KUKA KRL program: MyProgram_314().src

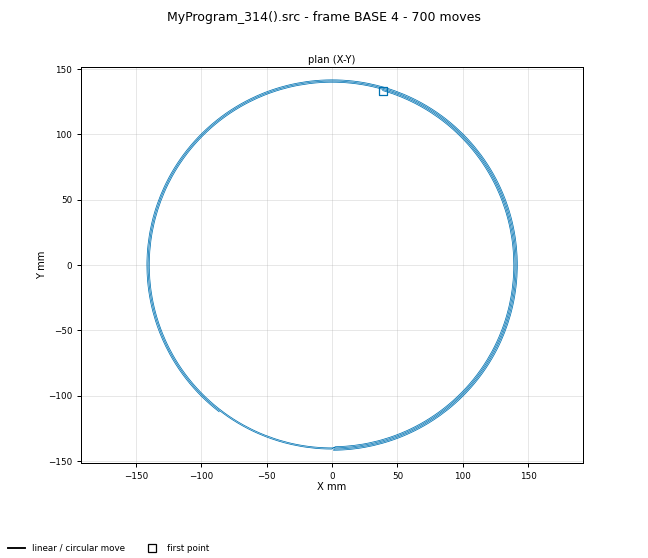
[picture p0: tool path of MyProgram_314().src in frame BASE 4, 700 of 700 moves have a stored position in this frame; points joined in program order, loops and branches not executed]
&ACCESS RVP
&REL 1
&PARAM TEMPLATE = C:\KRC\Roboter\Template\vorgabe
&PARAM EDITMASK = *
DEF MyProgram_314()
; ---- Setting reference (Base) ----
$BASE = BASE_DATA[4]

; --------------------------
; ---- Setting tool (TCP) ----
$TOOL = TOOL_DATA[3]
; --------------------------

$VEL.CP = VEL_APROX_PRINT
Startdeposition()
$VEL.CP = VEL_PRINT
LIN {X 38.6901,Y 133.5484,Z 183,A 74.6079,B 4.1647,C 0.0823,E1 4.2136,E2 378.5903} C_DIS
LIN {X 41.5849,Y 132.6771,Z 183,A 73.3895,B 4.1647,C 0.0831,E1 4.2168,E2 379.8051} C_DIS
LIN {X 46.4124,Y 131.0665,Z 183,A 71.2167,B 4.1647,C 0.0859,E1 4.2226,E2 381.9869} C_DIS
LIN {X 50.1301,Y 129.6879,Z 183,A 69.6295,B 4.1646,C 0.0872,E1 4.2267,E2 383.568} C_DIS
LIN {X 53.3488,Y 128.3973,Z 183,A 68.1306,B 4.1646,C 0.0895,E1 4.2306,E2 385.0754} C_DIS
LIN {X 57.8954,Y 126.4131,Z 183,A 65.4479,B 4.1643,C 0.0987,E1 4.2376,E2 387.8363} C_DIS
LIN {X 63.5941,Y 123.6447,Z 183,A 63.5677,B 4.1644,C 0.0945,E1 4.2421,E2 389.6266} C_DIS
LIN {X 67.8619,Y 121.3561,Z 183,A 61.634,B 4.1644,C 0.0967,E1 4.2468,E2 391.5526} C_DIS
LIN {X 71.8304,Y 119.0499,Z 183,A 59.745,B 4.1644,C 0.0995,E1 4.2513,E2 393.4412} C_DIS
LIN {X 75.3981,Y 116.8235,Z 183,A 58.2199,B 4.1644,C 0.1,E1 4.2549,E2 394.9405} C_DIS
LIN {X 81.6488,Y 112.543,Z 183,A 55.058,B 4.1642,C 0.1056,E1 4.2622,E2 398.1075} C_DIS
LIN {X 85.258,Y 109.8341,Z 183,A 53.2155,B 4.1641,C 0.1087,E1 4.2662,E2 399.948} C_DIS
LIN {X 88.7432,Y 107.0378,Z 183,A 51.4298,B 4.1641,C 0.1114,E1 4.2701,E2 401.727} C_DIS
LIN {X 92.1738,Y 104.0983,Z 183,A 49.6505,B 4.1639,C 0.114,E1 4.2738,E2 403.4963} C_DIS
LIN {X 95.5936,Y 100.9672,Z 183,A 47.5183,B 4.1638,C 0.1203,E1 4.2782,E2 405.6563} C_DIS
LIN {X 98.0318,Y 98.6013,Z 183,A 46.3699,B 4.1638,C 0.1203,E1 4.2805,E2 406.7736} C_DIS
LIN {X 101.2747,Y 95.2677,Z 183,A 44.4916,B 4.1637,C 0.1238,E1 4.2841,E2 408.6476} C_DIS
LIN {X 104.2938,Y 91.9527,Z 183,A 42.7466,B 4.1636,C 0.1266,E1 4.2873,E2 410.3801} C_DIS
LIN {X 107.0493,Y 88.7294,Z 183,A 41.1805,B 4.1636,C 0.1283,E1 4.2901,E2 411.9238} C_DIS
LIN {X 109.6954,Y 85.4369,Z 183,A 39.261,B 4.1633,C 0.1343,E1 4.2935,E2 413.8663} C_DIS
LIN {X 112.5064,Y 81.6994,Z 183,A 37.4355,B 4.1633,C 0.1375,E1 4.2965,E2 415.6797} C_DIS
LIN {X 115.0062,Y 78.1414,Z 183,A 35.6994,B 4.1631,C 0.1411,E1 4.2992,E2 417.4092} C_DIS
LIN {X 117.403,Y 74.4922,Z 183,A 33.895,B 4.163,C 0.1454,E1 4.302,E2 419.2149} C_DIS
LIN {X 119.858,Y 70.4735,Z 183,A 32.0698,B 4.1628,C 0.1488,E1 4.3046,E2 421.0263} C_DIS
LIN {X 121.9501,Y 66.7885,Z 183,A 30.3317,B 4.1627,C 0.153,E1 4.3069,E2 422.7641} C_DIS
LIN {X 123.8361,Y 63.2182,Z 183,A 28.7952,B 4.1626,C 0.1557,E1 4.3089,E2 424.285} C_DIS
LIN {X 125.6527,Y 59.5273,Z 183,A 27.0862,B 4.1624,C 0.1602,E1 4.311,E2 425.9966} C_DIS
LIN {X 127.4768,Y 55.5132,Z 183,A 25.4211,B 4.1624,C 0.1631,E1 4.3128,E2 427.6432} C_DIS
LIN {X 128.8068,Y 52.3534,Z 183,A 24.0226,B 4.1622,C 0.1666,E1 4.3143,E2 429.0406} C_DIS
LIN {X 130.1139,Y 49.0137,Z 183,A 22.5912,B 4.162,C 0.17,E1 4.3158,E2 430.4669} C_DIS
LIN {X 131.3645,Y 45.5554,Z 183,A 21.1712,B 4.162,C 0.1728,E1 4.3171,E2 431.8754} C_DIS
LIN {X 132.3962,Y 42.4643,Z 183,A 19.8538,B 4.1618,C 0.1762,E1 4.3182,E2 433.1903} C_DIS
LIN {X 133.3699,Y 39.2998,Z 183,A 18.6395,B 4.1618,C 0.178,E1 4.3192,E2 434.3862} C_DIS
LIN {X 134.5526,Y 35.0458,Z 183,A 16.6466,B 4.1614,C 0.1851,E1 4.3207,E2 436.4024} C_DIS
LIN {X 135.5223,Y 31.0755,Z 183,A 15.1454,B 4.1613,C 0.1875,E1 4.3216,E2 437.8811} C_DIS
LIN {X 136.2197,Y 27.8599,Z 183,A 13.8266,B 4.1611,C 0.1908,E1 4.3224,E2 439.1959} C_DIS
LIN {X 137.5207,Y 20.5096,Z 183,A 10.874,B 4.1608,C 0.1979,E1 4.3238,E2 442.1347} C_DIS
LIN {X 137.9086,Y 17.7021,Z 183,A 9.3425,B 4.1604,C 0.2057,E1 4.3243,E2 443.7134} C_DIS
LIN {X 138.3551,Y 13.7893,Z 183,A 8.0826,B 4.1604,C 0.2057,E1 4.3247,E2 444.9281} C_DIS
LIN {X 138.6565,Y 10.3177,Z 183,A 6.7452,B 4.1603,C 0.2086,E1 4.325,E2 446.2537} C_DIS
LIN {X 138.8833,Y 6.6033,Z 183,A 5.211,B 4.1601,C 0.2129,E1 4.3252,E2 447.7891} C_DIS
LIN {X 139.0156,Y 2.6101,Z 183,A 3.8011,B 4.16,C 0.2146,E1 4.3252,E2 449.1697} C_DIS
LIN {X 139.0434,Y -0.021,Z 183,A 2.504,B 4.1597,C 0.2204,E1 4.3253,E2 450.495} C_DIS
LIN {X 138.9836,Y -3.952,Z 183,A 1.081,B 4.1596,C 0.2225,E1 4.3253,E2 451.8937} C_DIS
LIN {X 138.8076,Y -8.0465,Z 183,A -0.5936,B 4.1593,C 0.2271,E1 4.325,E2 453.5677} C_DIS
LIN {X 138.5359,Y -11.8261,Z 183,A -2.0469,B 4.1591,C 0.2301,E1 4.3247,E2 455.0081} C_DIS
LIN {X 138.1515,Y -15.7085,Z 183,A -3.7013,B 4.1589,C 0.2353,E1 4.3242,E2 456.6699} C_DIS
LIN {X 137.76,Y -18.8356,Z 183,A -5.4114,B 4.1584,C 0.2441,E1 4.3235,E2 458.434} C_DIS
LIN {X 137.0345,Y -23.5365,Z 183,A -6.7142,B 4.1585,C 0.2414,E1 4.323,E2 459.6534} C_DIS
LIN {X 135.6633,Y -30.4582,Z 183,A -9.607,B 4.158,C 0.2493,E1 4.3214,E2 462.5467} C_DIS
LIN {X 134.9201,Y -33.5994,Z 183,A -11.0898,B 4.1577,C 0.2549,E1 4.3203,E2 464.0503} C_DIS
LIN {X 133.5628,Y -38.6411,Z 183,A -12.8026,B 4.1577,C 0.2553,E1 4.3191,E2 465.7078} C_DIS
LIN {X 132.6254,Y -41.7467,Z 183,A -14.2307,B 4.1574,C 0.2601,E1 4.3179,E2 467.1489} C_DIS
LIN {X 131.4955,Y -45.1776,Z 183,A -16.076,B 4.1569,C 0.2685,E1 4.3162,E2 469.0418} C_DIS
LIN {X 130.171,Y -48.8614,Z 183,A -17.2495,B 4.1569,C 0.2674,E1 4.3152,E2 470.1594} C_DIS
LIN {X 128.9622,Y -51.9679,Z 183,A -18.5228,B 4.1568,C 0.2698,E1 4.3139,E2 471.4208} C_DIS
LIN {X 127.7218,Y -54.9464,Z 183,A -19.807,B 4.1566,C 0.2728,E1 4.3125,E2 472.7002} C_DIS
LIN {X 125.9756,Y -58.8415,Z 183,A -21.66,B 4.1562,C 0.2785,E1 4.3103,E2 474.5669} C_DIS
LIN {X 124.2812,Y -62.3432,Z 183,A -23.2186,B 4.156,C 0.2821,E1 4.3084,E2 476.1211} C_DIS
LIN {X 122.3977,Y -65.9643,Z 183,A -24.8332,B 4.1557,C 0.2855,E1 4.3063,E2 477.7283} C_DIS
LIN {X 118.702,Y -72.4046,Z 183,A -27.8541,B 4.1552,C 0.2927,E1 4.302,E2 480.7467} C_DIS
LIN {X 116.1898,Y -76.3701,Z 183,A -29.6676,B 4.155,C 0.2959,E1 4.2993,E2 482.546} C_DIS
LIN {X 113.7481,Y -79.9617,Z 183,A -31.4516,B 4.1547,C 0.3001,E1 4.2965,E2 484.3308} C_DIS
LIN {X 111.0357,Y -83.6871,Z 183,A -33.2889,B 4.1544,C 0.3038,E1 4.2934,E2 486.1616} C_DIS
LIN {X 108.1883,Y -87.337,Z 183,A -35.1586,B 4.1541,C 0.3077,E1 4.2902,E2 488.0279} C_DIS
LIN {X 105.1296,Y -90.9963,Z 183,A -37.0564,B 4.1539,C 0.3112,E1 4.2868,E2 489.9184} C_DIS
LIN {X 102.0998,Y -94.3835,Z 183,A -38.8813,B 4.1536,C 0.3147,E1 4.2833,E2 491.7386} C_DIS
LIN {X 99.1255,Y -97.5019,Z 183,A -40.6699,B 4.1533,C 0.3186,E1 4.2799,E2 493.5304} C_DIS
LIN {X 95.672,Y -100.8932,Z 183,A -42.5669,B 4.1531,C 0.3215,E1 4.2761,E2 495.4161} C_DIS
LIN {X 92.5142,Y -103.7964,Z 183,A -44.2085,B 4.1529,C 0.3236,E1 4.2727,E2 497.0426} C_DIS
LIN {X 89.4317,Y -106.4633,Z 183,A -45.9892,B 4.1526,C 0.328,E1 4.2689,E2 498.838} C_DIS
LIN {X 85.6496,Y -109.5294,Z 183,A -47.8402,B 4.1524,C 0.3299,E1 4.2649,E2 500.6701} C_DIS
LIN {X 82.2654,Y -112.0931,Z 183,A -49.5595,B 4.1522,C 0.3327,E1 4.261,E2 502.3869} C_DIS
LIN {X 78.6574,Y -114.6537,Z 183,A -51.3807,B 4.152,C 0.3358,E1 4.2569,E2 504.2092} C_DIS
LIN {X 74.8249,Y -117.191,Z 183,A -53.2055,B 4.1518,C 0.3381,E1 4.2526,E2 506.0263} C_DIS
LIN {X 71.0409,Y -119.5227,Z 183,A -54.9847,B 4.1516,C 0.3404,E1 4.2484,E2 507.7999} C_DIS
LIN {X 67.9317,Y -121.3169,Z 183,A -56.5366,B 4.1513,C 0.3434,E1 4.2446,E2 509.3626} C_DIS
LIN {X 63.7821,Y -123.549,Z 183,A -58.4038,B 4.1512,C 0.3454,E1 4.24,E2 511.2214} C_DIS
LIN {X 60.2118,Y -125.3257,Z 183,A -59.9855,B 4.1511,C 0.3469,E1 4.236,E2 512.7961} C_DIS
LIN {X 57.1271,Y -126.7618,Z 183,A -61.3521,B 4.1509,C 0.3484,E1 4.2326,E2 514.159} C_DIS
LIN {X 52.8925,Y -128.5879,Z 183,A -63.2697,B 4.1507,C 0.3509,E1 4.2276,E2 516.0803} C_DIS
LIN {X 48.2273,Y -130.4085,Z 183,A -65.6657,B 4.1502,C 0.3568,E1 4.2212,E2 518.5216} C_DIS
LIN {X 44.2524,Y -131.8096,Z 183,A -66.9438,B 4.1505,C 0.3537,E1 4.218,E2 519.7401} C_DIS
LIN {X 41.1074,Y -132.8244,Z 183,A -68.3125,B 4.1504,C 0.3551,E1 4.2144,E2 521.1107} C_DIS
LIN {X 38.0143,Y -133.7431,Z 183,A -69.6747,B 4.1502,C 0.3566,E1 4.2107,E2 522.4781} C_DIS
LIN {X 34.8764,Y -134.596,Z 183,A -71.3347,B 4.1498,C 0.3611,E1 4.2061,E2 524.1815} C_DIS
LIN {X 31.0318,Y -135.5323,Z 183,A -72.5205,B 4.1501,C 0.3578,E1 4.203,E2 525.3093} C_DIS
LIN {X 27.8154,Y -136.2288,Z 183,A -73.7669,B 4.1501,C 0.3576,E1 4.1997,E2 526.5418} C_DIS
LIN {X 23.5961,Y -137.0246,Z 183,A -75.5986,B 4.15,C 0.3594,E1 4.1946,E2 528.383} C_DIS
LIN {X 16.847,Y -138.0157,Z 183,A -78.445,B 4.1498,C 0.3612,E1 4.1867,E2 531.2357} C_DIS
LIN {X 13.4116,Y -138.3913,Z 183,A -79.7844,B 4.1498,C 0.361,E1 4.183,E2 532.5645} C_DIS
LIN {X 10.2776,Y -138.6594,Z 183,A -81.1632,B 4.1498,C 0.3623,E1 4.1791,E2 533.9551} C_DIS
LIN {X 6.3212,Y -138.8975,Z 183,A -82.7609,B 4.1498,C 0.3624,E1 4.1747,E2 535.5489} C_DIS
LIN {X 2.5424,Y -139.0167,Z 183,A -84.3219,B 4.1498,C 0.3628,E1 4.1703,E2 537.111} C_DIS
LIN {X 2.5424,Y -139.0167,Z 183,A -84.3219,B 4.1498,C 0.3628,E1 4.1703,E2 537.111} C_DIS
Enddeposition()
LIN {X 0.9796,Y -139.9354,Z 183,A -84.7324,B 4.1032,C 0.3616,E1 4.1227,E2 537.5356} C_DIS
Startdeposition()
$VEL.CP = VEL_PRINT
LIN {X 3.736,Y -139.891,Z 183,A -83.0903,B 4.1037,C 0.3563,E1 4.1275,E2 535.8237} C_DIS
LIN {X 7.4249,Y -139.7442,Z 183,A -81.5162,B 4.1037,C 0.3553,E1 4.1319,E2 534.2403} C_DIS
LIN {X 11.7645,Y -139.4453,Z 183,A -79.8462,B 4.1037,C 0.3557,E1 4.1365,E2 532.5844} C_DIS
LIN {X 15.3477,Y -139.097,Z 183,A -78.4152,B 4.1037,C 0.3555,E1 4.1405,E2 531.1584} C_DIS
LIN {X 18.9985,Y -138.6472,Z 183,A -76.606,B 4.1041,C 0.3517,E1 4.1456,E2 529.3073} C_DIS
LIN {X 22.2848,Y -138.1565,Z 183,A -75.599,B 4.1038,C 0.3545,E1 4.1482,E2 528.3475} C_DIS
LIN {X 28.614,Y -136.9858,Z 183,A -72.9607,B 4.104,C 0.3528,E1 4.1555,E2 525.7073} C_DIS
LIN {X 31.4563,Y -136.3595,Z 183,A -71.592,B 4.1042,C 0.35,E1 4.1593,E2 524.3138} C_DIS
LIN {X 36.5456,Y -135.0851,Z 183,A -69.6426,B 4.1042,C 0.3503,E1 4.1645,E2 522.3901} C_DIS
LIN {X 39.5732,Y -134.2287,Z 183,A -68.346,B 4.1043,C 0.349,E1 4.168,E2 521.0915} C_DIS
LIN {X 43.4113,Y -133.0393,Z 183,A -66.4686,B 4.1047,C 0.3449,E1 4.1731,E2 519.1815} C_DIS
LIN {X 49.2904,Y -130.9725,Z 183,A -64.2268,B 4.1046,C 0.3455,E1 4.1788,E2 516.9799} C_DIS
LIN {X 52.381,Y -129.7671,Z 183,A -62.8427,B 4.1048,C 0.3436,E1 4.1824,E2 515.5914} C_DIS
LIN {X 55.7191,Y -128.3694,Z 183,A -61.4245,B 4.1048,C 0.3425,E1 4.1861,E2 514.1807} C_DIS
LIN {X 59.1512,Y -126.8251,Z 183,A -59.8958,B 4.105,C 0.3406,E1 4.19,E2 512.6526} C_DIS
LIN {X 62.3488,Y -125.2842,Z 183,A -58.4371,B 4.1052,C 0.3386,E1 4.1936,E2 511.192} C_DIS
LIN {X 66.3568,Y -123.2097,Z 183,A -56.3022,B 4.1057,C 0.3327,E1 4.199,E2 509.0168} C_DIS
LIN {X 69.5862,Y -121.4151,Z 183,A -55.0814,B 4.1056,C 0.3337,E1 4.2019,E2 507.8345} C_DIS
LIN {X 73.4646,Y -119.1087,Z 183,A -53.2489,B 4.1058,C 0.331,E1 4.2062,E2 506.0026} C_DIS
LIN {X 77.1485,Y -116.7561,Z 183,A -51.2986,B 4.1062,C 0.3262,E1 4.2109,E2 504.0291} C_DIS
LIN {X 79.9664,Y -114.8443,Z 183,A -49.7608,B 4.1065,C 0.3221,E1 4.2144,E2 502.4707} C_DIS
LIN {X 83.5364,Y -112.2742,Z 183,A -48.745,B 4.106,C 0.3281,E1 4.2165,E2 501.5598} C_DIS
LIN {X 87.4834,Y -109.2276,Z 183,A -46.0047,B 4.107,C 0.3161,E1 4.2227,E2 498.7234} C_DIS
LIN {X 90.836,Y -106.4551,Z 183,A -44.2671,B 4.1072,C 0.3132,E1 4.2264,E2 496.9903} C_DIS
LIN {X 94.111,Y -103.571,Z 183,A -42.8999,B 4.1071,C 0.3147,E1 4.2291,E2 495.6784} C_DIS
LIN {X 97.4757,Y -100.4109,Z 183,A -40.7399,B 4.1076,C 0.3076,E1 4.2335,E2 493.4803} C_DIS
LIN {X 100.3317,Y -97.5575,Z 183,A -39.3383,B 4.1076,C 0.3071,E1 4.2362,E2 492.1114} C_DIS
LIN {X 103.6153,Y -94.0622,Z 183,A -37.5343,B 4.1078,C 0.3048,E1 4.2396,E2 490.3272} C_DIS
LIN {X 106.5619,Y -90.7105,Z 183,A -35.7303,B 4.1081,C 0.3011,E1 4.2429,E2 488.5248} C_DIS
LIN {X 108.8719,Y -87.9247,Z 183,A -34.301,B 4.1083,C 0.2984,E1 4.2454,E2 487.1013} C_DIS
LIN {X 111.7372,Y -84.2533,Z 183,A -32.4639,B 4.1085,C 0.2948,E1 4.2485,E2 485.272} C_DIS
LIN {X 114.4356,Y -80.5502,Z 183,A -30.6302,B 4.1088,C 0.2909,E1 4.2515,E2 483.4424} C_DIS
LIN {X 117.0012,Y -76.7762,Z 183,A -28.8143,B 4.1091,C 0.2871,E1 4.2543,E2 481.632} C_DIS
LIN {X 119.43,Y -72.941,Z 183,A -26.8652,B 4.1095,C 0.2814,E1 4.2572,E2 479.6691} C_DIS
LIN {X 122.7694,Y -67.168,Z 183,A -24.2566,B 4.1098,C 0.2761,E1 4.2607,E2 477.0746} C_DIS
LIN {X 124.8058,Y -63.2994,Z 183,A -22.7216,B 4.1099,C 0.2746,E1 4.2627,E2 475.5722} C_DIS
LIN {X 126.202,Y -60.4677,Z 183,A -21.0647,B 4.1105,C 0.2668,E1 4.2647,E2 473.8654} C_DIS
LIN {X 127.8914,Y -56.8084,Z 183,A -19.8668,B 4.1104,C 0.2681,E1 4.266,E2 472.7267} C_DIS
LIN {X 129.2282,Y -53.6973,Z 183,A -18.5019,B 4.1106,C 0.2647,E1 4.2675,E2 471.3635} C_DIS
LIN {X 130.534,Y -50.4403,Z 183,A -17.1692,B 4.1107,C 0.2622,E1 4.2688,E2 470.0435} C_DIS
LIN {X 132.5502,Y -44.8802,Z 183,A -14.7377,B 4.1112,C 0.2556,E1 4.2711,E2 467.6087} C_DIS
LIN {X 133.7534,Y -41.1506,Z 183,A -13.1595,B 4.1114,C 0.2515,E1 4.2724,E2 466.0326} C_DIS
LIN {X 134.9002,Y -37.222,Z 183,A -10.8806,B 4.1121,C 0.2393,E1 4.2742,E2 463.6718} C_DIS
LIN {X 136.3491,Y -31.5022,Z 183,A -9.3294,B 4.1119,C 0.2435,E1 4.2751,E2 462.2341} C_DIS
LIN {X 137.6457,Y -25.2466,Z 183,A -6.8343,B 4.1122,C 0.2378,E1 4.2765,E2 459.7531} C_DIS
LIN {X 138.1132,Y -22.5464,Z 183,A -5.5729,B 4.1125,C 0.2329,E1 4.2771,E2 458.4724} C_DIS
LIN {X 138.6569,Y -18.9261,Z 183,A -4.2506,B 4.1126,C 0.2309,E1 4.2776,E2 457.1723} C_DIS
LIN {X 139.1517,Y -14.8395,Z 183,A -2.5527,B 4.1129,C 0.226,E1 4.2781,E2 455.4715} C_DIS
LIN {X 139.5467,Y -10.4986,Z 183,A -0.8139,B 4.1131,C 0.2215,E1 4.2785,E2 453.7373} C_DIS
LIN {X 139.7795,Y -6.7232,Z 183,A 0.6384,B 4.1133,C 0.2183,E1 4.2788,E2 452.2967} C_DIS
LIN {X 139.8999,Y -3.4143,Z 183,A 2.0229,B 4.1135,C 0.2141,E1 4.2788,E2 450.9073} C_DIS
LIN {X 139.9405,Y 0.6341,Z 183,A 3.6219,B 4.1137,C 0.2102,E1 4.2788,E2 449.315} C_DIS
LIN {X 139.8518,Y 5.0079,Z 183,A 5.3432,B 4.1139,C 0.206,E1 4.2788,E2 447.6016} C_DIS
LIN {X 139.658,Y 8.895,Z 183,A 6.8354,B 4.1141,C 0.2027,E1 4.2785,E2 446.1216} C_DIS
LIN {X 139.3232,Y 13.1336,Z 183,A 8.5685,B 4.1143,C 0.1979,E1 4.2781,E2 444.3883} C_DIS
LIN {X 138.769,Y 18.0706,Z 183,A 10.4614,B 4.1145,C 0.194,E1 4.2775,E2 442.5126} C_DIS
LIN {X 138.2844,Y 21.4663,Z 183,A 12.454,B 4.115,C 0.1827,E1 4.2766,E2 440.4419} C_DIS
LIN {X 137.365,Y 26.7287,Z 183,A 14.253,B 4.115,C 0.1815,E1 4.2757,E2 438.6927} C_DIS
LIN {X 136.6393,Y 30.2249,Z 183,A 15.3384,B 4.115,C 0.1821,E1 4.2751,E2 437.6557} C_DIS
LIN {X 135.9274,Y 33.2762,Z 183,A 16.5818,B 4.1152,C 0.1791,E1 4.2742,E2 436.4166} C_DIS
LIN {X 134.5668,Y 38.4144,Z 183,A 18.6873,B 4.1154,C 0.174,E1 4.2727,E2 434.3192} C_DIS
LIN {X 133.7792,Y 41.0662,Z 183,A 19.8093,B 4.1155,C 0.171,E1 4.2718,E2 433.198} C_DIS
LIN {X 132.7549,Y 44.2656,Z 183,A 21.1119,B 4.1157,C 0.1682,E1 4.2707,E2 431.9041} C_DIS
LIN {X 131.6037,Y 47.579,Z 183,A 22.5424,B 4.1158,C 0.1645,E1 4.2693,E2 430.4736} C_DIS
LIN {X 130.3743,Y 50.8513,Z 183,A 23.9233,B 4.1159,C 0.1613,E1 4.268,E2 429.0985} C_DIS
LIN {X 129.0654,Y 54.0872,Z 183,A 25.3216,B 4.1161,C 0.1579,E1 4.2665,E2 427.7035} C_DIS
LIN {X 127.6068,Y 57.4446,Z 183,A 26.7566,B 4.1161,C 0.1548,E1 4.2649,E2 426.2761} C_DIS
LIN {X 126.1331,Y 60.6118,Z 183,A 28.142,B 4.1163,C 0.1517,E1 4.2632,E2 424.8959} C_DIS
LIN {X 124.5227,Y 63.8554,Z 183,A 29.5799,B 4.1164,C 0.1485,E1 4.2614,E2 423.4631} C_DIS
LIN {X 122.717,Y 67.2641,Z 183,A 31.2028,B 4.1166,C 0.144,E1 4.2593,E2 421.834} C_DIS
LIN {X 120.4869,Y 71.1818,Z 183,A 32.974,B 4.1167,C 0.1403,E1 4.2568,E2 420.0718} C_DIS
LIN {X 118.1588,Y 74.983,Z 183,A 34.7723,B 4.1168,C 0.1363,E1 4.2541,E2 418.2762} C_DIS
LIN {X 115.6435,Y 78.8073,Z 183,A 36.5684,B 4.117,C 0.1327,E1 4.2514,E2 416.4896} C_DIS
LIN {X 113.0942,Y 82.4236,Z 183,A 38.3345,B 4.117,C 0.1291,E1 4.2485,E2 414.7287} C_DIS
LIN {X 110.4665,Y 85.9129,Z 183,A 40.5753,B 4.1174,C 0.1197,E1 4.2446,E2 412.4291} C_DIS
LIN {X 107.2942,Y 89.8431,Z 183,A 42.0484,B 4.1173,C 0.1221,E1 4.2421,E2 411.0322} C_DIS
LIN {X 104.498,Y 93.0813,Z 183,A 43.8953,B 4.1174,C 0.1172,E1 4.2386,E2 409.1727} C_DIS
LIN {X 101.654,Y 96.1786,Z 183,A 45.463,B 4.1174,C 0.1154,E1 4.2357,E2 407.6243} C_DIS
LIN {X 98.5993,Y 99.3076,Z 183,A 47.8184,B 4.1177,C 0.1053,E1 4.2309,E2 405.196} C_DIS
LIN {X 94.5364,Y 103.1831,Z 183,A 49.3534,B 4.1177,C 0.1095,E1 4.2279,E2 403.7587} C_DIS
LIN {X 92.1545,Y 105.3158,Z 183,A 50.7655,B 4.1177,C 0.1058,E1 4.2249,E2 402.3333} C_DIS
LIN {X 88.3263,Y 108.5466,Z 183,A 52.7567,B 4.1178,C 0.1027,E1 4.2207,E2 400.3495} C_DIS
LIN {X 84.6897,Y 111.4076,Z 183,A 54.6308,B 4.1178,C 0.0996,E1 4.2165,E2 398.4779} C_DIS
LIN {X 80.7626,Y 114.2855,Z 183,A 56.794,B 4.118,C 0.0943,E1 4.2116,E2 396.2929} C_DIS
LIN {X 77.8149,Y 116.3129,Z 183,A 57.9478,B 4.118,C 0.0953,E1 4.209,E2 395.1787} C_DIS
LIN {X 74.2993,Y 118.5902,Z 183,A 59.7134,B 4.118,C 0.0921,E1 4.2048,E2 393.4066} C_DIS
LIN {X 70.6261,Y 120.8133,Z 183,A 61.3857,B 4.118,C 0.0904,E1 4.2008,E2 391.7453} C_DIS
LIN {X 66.6812,Y 123.0349,Z 183,A 63.2276,B 4.1182,C 0.0879,E1 4.1963,E2 389.9049} C_DIS
LIN {X 62.8771,Y 125.0208,Z 183,A 65.1802,B 4.1182,C 0.0834,E1 4.1914,E2 387.9276} C_DIS
LIN {X 59.7314,Y 126.5537,Z 183,A 66.2498,B 4.1182,C 0.0854,E1 4.1888,E2 386.9042} C_DIS
LIN {X 57.0233,Y 127.7953,Z 183,A 67.4511,B 4.1182,C 0.0841,E1 4.1858,E2 385.7053} C_DIS
LIN {X 53.6698,Y 129.2397,Z 183,A 68.9309,B 4.1182,C 0.0825,E1 4.182,E2 384.2277} C_DIS
LIN {X 50.4125,Y 130.5449,Z 183,A 70.3823,B 4.1182,C 0.0808,E1 4.1782,E2 382.7746} C_DIS
LIN {X 46.7659,Y 131.8969,Z 183,A 72.6408,B 4.1185,C 0.0724,E1 4.172,E2 380.4319} C_DIS
LIN {X 41.4513,Y 133.6614,Z 183,A 74.0818,B 4.1183,C 0.0789,E1 4.1685,E2 379.0994} C_DIS
LIN {X 38.9881,Y 134.4,Z 183,A 75.2244,B 4.1183,C 0.0771,E1 4.1654,E2 377.9458} C_DIS
LIN {X 35.4655,Y 135.3732,Z 183,A 76.9224,B 4.1184,C 0.0739,E1 4.1607,E2 376.2226} C_DIS
LIN {X 31.1573,Y 136.4278,Z 183,A 78.8391,B 4.1184,C 0.0716,E1 4.1555,E2 374.2936} C_DIS
LIN {X 27.7717,Y 137.1572,Z 183,A 79.9625,B 4.1184,C 0.0735,E1 4.1525,E2 373.2078} C_DIS
LIN {X 23.9362,Y 137.8802,Z 183,A 81.8001,B 4.1184,C 0.0703,E1 4.1474,E2 371.3406} C_DIS
LIN {X 18.614,Y 138.6978,Z 183,A 83.5571,B 4.1184,C 0.0735,E1 4.1427,E2 369.6406} C_DIS
LIN {X 14.7295,Y 139.1635,Z 183,A 85.3706,B 4.1184,C 0.0709,E1 4.1376,E2 367.8011} C_DIS
LIN {X 10.3429,Y 139.558,Z 183,A 87.1238,B 4.1184,C 0.0709,E1 4.1327,E2 366.0549} C_DIS
LIN {X 6.8393,Y 139.7736,Z 183,A 88.5411,B 4.1184,C 0.0707,E1 4.1288,E2 364.6407} C_DIS
LIN {X 2.8571,Y 139.9126,Z 183,A 90.2468,B 4.1184,C 0.0697,E1 4.124,E2 362.9263} C_DIS
LIN {X -1.1552,Y 139.9366,Z 183,A 91.7864,B 4.1184,C 0.0705,E1 4.1197,E2 361.4004} C_DIS
LIN {X -4.9256,Y 139.855,Z 183,A 93.4859,B 4.1185,C 0.0691,E1 4.1149,E2 359.6821} C_DIS
LIN {X -8.937,Y 139.6555,Z 183,A 95.167,B 4.1185,C 0.069,E1 4.1102,E2 357.9971} C_DIS
LIN {X -12.5685,Y 139.3774,Z 183,A 96.6629,B 4.1185,C 0.0692,E1 4.106,E2 356.5014} C_DIS
LIN {X -16.9807,Y 138.9072,Z 183,A 98.3677,B 4.1185,C 0.0706,E1 4.1013,E2 354.8115} C_DIS
LIN {X -25.8176,Y 137.5391,Z 183,A 102.1653,B 4.1185,C 0.0709,E1 4.0908,E2 350.9989} C_DIS
LIN {X -30.0571,Y 136.6755,Z 183,A 103.765,B 4.1185,C 0.0732,E1 4.0865,E2 349.4219} C_DIS
LIN {X -33.2613,Y 135.931,Z 183,A 105.2627,B 4.1185,C 0.0727,E1 4.0824,E2 347.906} C_DIS
LIN {X -39.3908,Y 134.2821,Z 183,A 107.7715,B 4.1185,C 0.0753,E1 4.0757,E2 345.41} C_DIS
LIN {X -42.9264,Y 133.1944,Z 183,A 109.3105,B 4.1184,C 0.0762,E1 4.0716,E2 343.869} C_DIS
LIN {X -47.7378,Y 131.5465,Z 183,A 111.7736,B 4.1184,C 0.075,E1 4.065,E2 341.3592} C_DIS
LIN {X -51.447,Y 130.1427,Z 183,A 113.3392,B 4.1184,C 0.077,E1 4.0609,E2 339.8021} C_DIS
LIN {X -54.5426,Y 128.8752,Z 183,A 114.3914,B 4.1183,C 0.081,E1 4.0583,E2 338.7908} C_DIS
LIN {X -57.2838,Y 127.6788,Z 183,A 115.6778,B 4.1183,C 0.0818,E1 4.055,E2 337.4974} C_DIS
LIN {X -63.1163,Y 124.899,Z 183,A 118.178,B 4.1182,C 0.086,E1 4.0488,E2 335.0173} C_DIS
LIN {X -66.457,Y 123.1559,Z 183,A 120.0042,B 4.1182,C 0.0858,E1 4.0442,E2 333.1567} C_DIS
LIN {X -70.4556,Y 120.9132,Z 183,A 121.9421,B 4.1182,C 0.0879,E1 4.0395,E2 331.2124} C_DIS
LIN {X -74.3908,Y 118.5325,Z 183,A 123.8402,B 4.1181,C 0.0905,E1 4.0349,E2 329.3138} C_DIS
LIN {X -78.1332,Y 116.0998,Z 183,A 125.6998,B 4.1181,C 0.093,E1 4.0306,E2 327.4515} C_DIS
LIN {X -81.8067,Y 113.5414,Z 183,A 127.5751,B 4.118,C 0.0956,E1 4.0263,E2 325.5723} C_DIS
LIN {X -85.4323,Y 110.839,Z 183,A 129.4921,B 4.118,C 0.0982,E1 4.022,E2 323.6484} C_DIS
LIN {X -89.045,Y 107.9578,Z 183,A 131.4149,B 4.1178,C 0.1013,E1 4.0179,E2 321.7231} C_DIS
LIN {X -92.5027,Y 105.0102,Z 183,A 133.2876,B 4.1178,C 0.1046,E1 4.0139,E2 319.8504} C_DIS
LIN {X -95.7881,Y 102.0224,Z 183,A 135.1861,B 4.1177,C 0.1075,E1 4.01,E2 317.943} C_DIS
LIN {X -99.1106,Y 98.7976,Z 183,A 137.1033,B 4.1176,C 0.111,E1 4.0062,E2 316.0246} C_DIS
LIN {X -102.1715,Y 95.6291,Z 183,A 138.9803,B 4.1176,C 0.1142,E1 4.0026,E2 314.1398} C_DIS
LIN {X -105.2561,Y 92.2229,Z 183,A 140.8656,B 4.1174,C 0.1181,E1 3.9991,E2 312.2555} C_DIS
LIN {X -108.1261,Y 88.8409,Z 183,A 142.7398,B 4.1173,C 0.1216,E1 3.9957,E2 310.3755} C_DIS
LIN {X -110.9074,Y 85.3437,Z 183,A 144.6571,B 4.1172,C 0.125,E1 3.9924,E2 308.4485} C_DIS
LIN {X -113.6937,Y 81.5943,Z 183,A 146.6929,B 4.1171,C 0.1285,E1 3.989,E2 306.3986} C_DIS
LIN {X -116.1425,Y 78.0699,Z 183,A 148.7842,B 4.1171,C 0.1304,E1 3.9857,E2 304.266} C_DIS
LIN {X -118.4609,Y 74.5042,Z 183,A 149.9556,B 4.1168,C 0.1383,E1 3.984,E2 303.1688} C_DIS
LIN {X -120.1572,Y 71.7362,Z 183,A 151.6342,B 4.1168,C 0.1392,E1 3.9816,E2 301.4468} C_DIS
LIN {X -122.3846,Y 67.8663,Z 183,A 153.3043,B 4.1165,C 0.1447,E1 3.9793,E2 299.7983} C_DIS
LIN {X -124.1581,Y 64.5626,Z 183,A 154.9275,B 4.1165,C 0.148,E1 3.9771,E2 298.1652} C_DIS
LIN {X -125.6226,Y 61.6627,Z 183,A 156.3336,B 4.1163,C 0.1509,E1 3.9754,E2 296.7504} C_DIS
LIN {X -127.221,Y 58.295,Z 183,A 157.8798,B 4.1162,C 0.1546,E1 3.9736,E2 295.2029} C_DIS
LIN {X -128.5896,Y 55.2098,Z 183,A 159.3132,B 4.1161,C 0.1579,E1 3.972,E2 293.764} C_DIS
LIN {X -129.954,Y 51.9174,Z 183,A 160.8333,B 4.1159,C 0.1613,E1 3.9704,E2 292.2373} C_DIS
LIN {X -131.1543,Y 48.8051,Z 183,A 162.2521,B 4.1159,C 0.1646,E1 3.9689,E2 290.8128} C_DIS
LIN {X -132.3351,Y 45.5065,Z 183,A 163.7053,B 4.1157,C 0.1683,E1 3.9676,E2 289.3584} C_DIS
LIN {X -133.3922,Y 42.3073,Z 183,A 165.1275,B 4.1155,C 0.1718,E1 3.9664,E2 287.9317} C_DIS
LIN {X -134.3663,Y 39.1031,Z 183,A 166.5616,B 4.1154,C 0.1751,E1 3.9652,E2 286.4907} C_DIS
LIN {X -135.2625,Y 35.8806,Z 183,A 168.0104,B 4.1152,C 0.1784,E1 3.9642,E2 285.0327} C_DIS
LIN {X -136.2165,Y 32.0771,Z 183,A 170.0127,B 4.1152,C 0.1803,E1 3.9628,E2 282.9805} C_DIS
LIN {X -137.0043,Y 28.5228,Z 183,A 171.1016,B 4.1149,C 0.1869,E1 3.9622,E2 281.9446} C_DIS
LIN {X -137.5553,Y 25.7329,Z 183,A 172.3639,B 4.1147,C 0.1896,E1 3.9616,E2 280.6706} C_DIS
LIN {X -138.1013,Y 22.6179,Z 183,A 174.1816,B 4.1147,C 0.19,E1 3.9607,E2 278.7862} C_DIS
LIN {X -138.7031,Y 18.5734,Z 183,A 175.5441,B 4.1144,C 0.1966,E1 3.9602,E2 277.4655} C_DIS
LIN {X -139.5417,Y 10.567,Z 183,A 178.704,B 4.1139,C 0.2067,E1 3.9594,E2 274.3258} C_DIS
LIN {X -139.8948,Y 3.5992,Z 183,A -178.298,B 4.1135,C 0.214,E1 3.959,E2 271.3117} C_DIS
LIN {X -139.924,Y -2.1731,Z 183,A -175.9702,B 4.1132,C 0.2209,E1 3.959,E2 268.9903} C_DIS
LIN {X -139.5576,Y -10.3491,Z 183,A -172.4354,B 4.1127,C 0.2292,E1 3.9594,E2 265.4342} C_DIS
LIN {X -138.9825,Y -16.3489,Z 183,A -169.6687,B 4.1124,C 0.2343,E1 3.9602,E2 262.6303} C_DIS
LIN {X -138.52,Y -19.8897,Z 183,A -167.5066,B 4.1124,C 0.234,E1 3.9611,E2 260.3773} C_DIS
LIN {X -137.6826,Y -25.0401,Z 183,A -165.9774,B 4.1119,C 0.2438,E1 3.9618,E2 258.9293} C_DIS
LIN {X -137.0047,Y -28.5212,Z 183,A -164.3296,B 4.1117,C 0.2465,E1 3.9627,E2 257.2567} C_DIS
LIN {X -136.0875,Y -32.6123,Z 183,A -162.6536,B 4.1114,C 0.2515,E1 3.9637,E2 255.587} C_DIS
LIN {X -135.245,Y -35.9462,Z 183,A -161.1804,B 4.1112,C 0.2549,E1 3.9648,E2 254.106} C_DIS
LIN {X -134.2335,Y -39.5566,Z 183,A -159.555,B 4.111,C 0.2585,E1 3.966,E2 252.4696} C_DIS
LIN {X -132.806,Y -44.1121,Z 183,A -157.0509,B 4.1109,C 0.2601,E1 3.9683,E2 249.8939} C_DIS
LIN {X -131.2476,Y -48.5558,Z 183,A -155.1072,B 4.1106,C 0.2651,E1 3.9702,E2 247.9492} C_DIS
LIN {X -129.6826,Y -52.5908,Z 183,A -153.7567,B 4.1101,C 0.2725,E1 3.9715,E2 246.6553} C_DIS
LIN {X -127.5452,Y -57.5824,Z 183,A -151.4832,B 4.1097,C 0.2778,E1 3.9741,E2 244.3763} C_DIS
LIN {X -126.1365,Y -60.6048,Z 183,A -150.0535,B 4.1095,C 0.2809,E1 3.9758,E2 242.9386} C_DIS
LIN {X -124.5684,Y -63.7657,Z 183,A -148.5489,B 4.1093,C 0.284,E1 3.9777,E2 241.4267} C_DIS
LIN {X -121.8164,Y -68.8812,Z 183,A -145.9084,B 4.109,C 0.2881,E1 3.9813,E2 238.7524} C_DIS
LIN {X -119.9839,Y -72.027,Z 183,A -144.4698,B 4.1087,C 0.292,E1 3.9833,E2 237.3214} C_DIS
LIN {X -117.588,Y -75.8751,Z 183,A -142.5575,B 4.1085,C 0.2959,E1 3.9862,E2 235.4022} C_DIS
LIN {X -115.0388,Y -79.6868,Z 183,A -140.6331,B 4.1082,C 0.2999,E1 3.9892,E2 233.4722} C_DIS
LIN {X -112.3686,Y -83.4096,Z 183,A -138.7009,B 4.1079,C 0.3037,E1 3.9924,E2 231.533} C_DIS
LIN {X -109.5261,Y -87.1083,Z 183,A -136.7696,B 4.1076,C 0.3076,E1 3.9958,E2 229.5993} C_DIS
LIN {X -106.6364,Y -90.6229,Z 183,A -134.8493,B 4.1073,C 0.3111,E1 3.9992,E2 227.6719} C_DIS
LIN {X -103.5646,Y -94.118,Z 183,A -132.9097,B 4.1071,C 0.3148,E1 4.0028,E2 225.7281} C_DIS
LIN {X -100.4903,Y -97.3936,Z 183,A -130.9986,B 4.1068,C 0.3179,E1 4.0065,E2 223.8077} C_DIS
LIN {X -97.1709,Y -100.706,Z 183,A -129.0664,B 4.1065,C 0.3214,E1 4.0104,E2 221.8742} C_DIS
LIN {X -93.9123,Y -103.7513,Z 183,A -127.1838,B 4.1063,C 0.3243,E1 4.0143,E2 219.9844} C_DIS
LIN {X -90.5224,Y -106.7218,Z 183,A -125.295,B 4.1061,C 0.3273,E1 4.0183,E2 218.0899} C_DIS
LIN {X -86.9058,Y -109.6873,Z 183,A -123.3232,B 4.1059,C 0.33,E1 4.0226,E2 216.1106} C_DIS
LIN {X -82.234,Y -113.2309,Z 183,A -120.5809,B 4.1058,C 0.3312,E1 4.0288,E2 213.3224} C_DIS
LIN {X -79.0283,Y -115.492,Z 183,A -119.3013,B 4.1054,C 0.3362,E1 4.0317,E2 212.0869} C_DIS
LIN {X -75.5193,Y -117.8163,Z 183,A -117.4912,B 4.1052,C 0.338,E1 4.0359,E2 210.2652} C_DIS
LIN {X -71.5769,Y -120.2522,Z 183,A -115.5812,B 4.105,C 0.3404,E1 4.0405,E2 208.3534} C_DIS
LIN {X -67.5868,Y -122.5394,Z 183,A -113.49,B 4.105,C 0.3411,E1 4.0457,E2 206.2339} C_DIS
LIN {X -61.7662,Y -125.5716,Z 183,A -111.0317,B 4.1045,C 0.3462,E1 4.0517,E2 203.8063} C_DIS
LIN {X -58.8063,Y -126.9846,Z 183,A -109.5381,B 4.1045,C 0.3463,E1 4.0556,E2 202.2921} C_DIS
LIN {X -55.1594,Y -128.6113,Z 183,A -107.9911,B 4.1043,C 0.3487,E1 4.0595,E2 200.7568} C_DIS
LIN {X -51.3998,Y -130.1611,Z 183,A -106.1964,B 4.1043,C 0.3492,E1 4.0642,E2 198.9444} C_DIS
LIN {X -44.1416,Y -132.7962,Z 183,A -103.462,B 4.1037,C 0.3555,E1 4.0712,E2 196.2671} C_DIS
LIN {X -40.0847,Y -134.0789,Z 183,A -101.2194,B 4.104,C 0.3523,E1 4.0774,E2 193.9566} C_DIS
LIN {X -33.7544,Y -135.8103,Z 183,A -98.6781,B 4.1038,C 0.3552,E1 4.0842,E2 191.4343} C_DIS
LIN {X -30.9039,Y -136.4857,Z 183,A -97.438,B 4.1038,C 0.3554,E1 4.0876,E2 190.1882} C_DIS
LIN {X -26.9919,Y -137.3147,Z 183,A -95.6214,B 4.1038,C 0.3545,E1 4.0926,E2 188.3469} C_DIS
LIN {X -22.3155,Y -138.1517,Z 183,A -93.7225,B 4.1038,C 0.3556,E1 4.0979,E2 186.4536} C_DIS
LIN {X -18.1788,Y -138.7548,Z 183,A -92.104,B 4.1036,C 0.3569,E1 4.1023,E2 184.8471} C_DIS
LIN {X -14.3131,Y -139.2083,Z 183,A -90.4674,B 4.1036,C 0.3567,E1 4.1069,E2 183.204} C_DIS
LIN {X -10.3014,Y -139.5611,Z 183,A -88.8774,B 4.1036,C 0.3574,E1 4.1113,E2 181.6213} C_DIS
LIN {X -6.698,Y -139.7807,Z 183,A -87.3381,B 4.1036,C 0.3568,E1 4.1156,E2 180.0731} C_DIS
LIN {X -2.4452,Y -139.9195,Z 183,A -85.6179,B 4.1036,C 0.3569,E1 4.1204,E2 178.355} C_DIS
LIN {X 0.9796,Y -139.9354,Z 183,A -84.7296,B 4.1032,C 0.3618,E1 4.1227,E2 177.5355} C_DIS
Enddeposition()
LIN {X 0.9796,Y -139.9354,Z 183,A -84.7296,B 4.1032,C 0.3618,E1 4.1227,E2 177.5355} C_DIS
Startdeposition()
$VEL.CP = VEL_PRINT
LIN {X -0.3233,Y -140.8422,Z 183,A -85.3433,B 3.9353,C 0.3599,E1 3.9532,E2 178.2404} C_DIS
LIN {X -4.3653,Y -140.7749,Z 183,A -87.0407,B 3.9353,C 0.3605,E1 3.9485,E2 179.9457} C_DIS
LIN {X -8.5637,Y -140.5812,Z 183,A -88.6536,B 3.9353,C 0.3596,E1 3.944,E2 181.5461} C_DIS
LIN {X -12.735,Y -140.2666,Z 183,A -90.419,B 3.9353,C 0.36,E1 3.9391,E2 183.3209} C_DIS
LIN {X -16.5443,Y -139.8666,Z 183,A -91.8728,B 3.9354,C 0.3588,E1 3.9351,E2 184.7612} C_DIS
LIN {X -19.8094,Y -139.4416,Z 183,A -93.2325,B 3.9354,C 0.3587,E1 3.9313,E2 186.124} C_DIS
LIN {X -23.809,Y -138.816,Z 183,A -94.9372,B 3.9354,C 0.3587,E1 3.9266,E2 187.8372} C_DIS
LIN {X -27.808,Y -138.0693,Z 183,A -96.5401,B 3.9356,C 0.3576,E1 3.9222,E2 189.4336} C_DIS
LIN {X -30.9784,Y -137.393,Z 183,A -97.9408,B 3.9356,C 0.3576,E1 3.9183,E2 190.8458} C_DIS
LIN {X -34.027,Y -136.6707,Z 183,A -99.0716,B 3.9357,C 0.3558,E1 3.9153,E2 191.9575} C_DIS
LIN {X -36.4124,Y -136.0532,Z 183,A -100.3953,B 3.9355,C 0.3579,E1 3.9116,E2 193.3248} C_DIS
LIN {X -41.0459,Y -134.7277,Z 183,A -102.0825,B 3.9359,C 0.3543,E1 3.9072,E2 194.9757} C_DIS
LIN {X -46.3752,Y -132.9875,Z 183,A -104.5091,B 3.9359,C 0.3538,E1 3.9007,E2 197.4225} C_DIS
LIN {X -50.6822,Y -131.4067,Z 183,A -106.3228,B 3.9361,C 0.3518,E1 3.896,E2 199.2295} C_DIS
LIN {X -53.9736,Y -130.0893,Z 183,A -107.7102,B 3.9362,C 0.35,E1 3.8924,E2 200.6097} C_DIS
LIN {X -56.5937,Y -128.9729,Z 183,A -109.0895,B 3.9362,C 0.3506,E1 3.8888,E2 202.019} C_DIS
LIN {X -60.2512,Y -127.304,Z 183,A -110.6339,B 3.9364,C 0.3481,E1 3.8849,E2 203.5513} C_DIS
LIN {X -63.5349,Y -125.6969,Z 183,A -111.9646,B 3.9367,C 0.3452,E1 3.8816,E2 204.861} C_DIS
LIN {X -68.2165,Y -123.2206,Z 183,A -114.3819,B 3.9367,C 0.3447,E1 3.8756,E2 207.314} C_DIS
LIN {X -71.9125,Y -121.1011,Z 183,A -116.2028,B 3.9368,C 0.3431,E1 3.8712,E2 209.1467} C_DIS
LIN {X -76.2205,Y -118.4372,Z 183,A -118.2903,B 3.9371,C 0.3404,E1 3.8662,E2 211.238} C_DIS
LIN {X -80.0511,Y -115.8828,Z 183,A -120.193,B 3.9373,C 0.3378,E1 3.8618,E2 213.1446} C_DIS
LIN {X -85.769,Y -111.7164,Z 183,A -123.1194,B 3.9377,C 0.3337,E1 3.8552,E2 216.0774} C_DIS
LIN {X -89.3977,Y -108.8347,Z 183,A -125.0442,B 3.9379,C 0.3308,E1 3.851,E2 218.0074} C_DIS
LIN {X -92.8134,Y -105.9366,Z 183,A -126.8942,B 3.9381,C 0.3278,E1 3.8471,E2 219.8608} C_DIS
LIN {X -96.2104,Y -102.8614,Z 183,A -128.8287,B 3.9384,C 0.3249,E1 3.8431,E2 221.8046} C_DIS
LIN {X -99.2843,Y -99.8972,Z 183,A -130.5606,B 3.9387,C 0.3216,E1 3.8396,E2 223.5354} C_DIS
LIN {X -102.1717,Y -96.9428,Z 183,A -132.3562,B 3.9389,C 0.3191,E1 3.8361,E2 225.3461} C_DIS
LIN {X -105.2779,Y -93.5602,Z 183,A -134.279,B 3.9391,C 0.3157,E1 3.8325,E2 227.2757} C_DIS
LIN {X -108.278,Y -90.0711,Z 183,A -136.2017,B 3.9394,C 0.3121,E1 3.829,E2 229.2047} C_DIS
LIN {X -111.1929,Y -86.4466,Z 183,A -138.1349,B 3.9397,C 0.3083,E1 3.8257,E2 231.1429} C_DIS
LIN {X -113.869,Y -82.89,Z 183,A -140.0047,B 3.94,C 0.3047,E1 3.8226,E2 233.02} C_DIS
LIN {X -116.5292,Y -79.1063,Z 183,A -141.917,B 3.9403,C 0.3006,E1 3.8195,E2 234.9358} C_DIS
LIN {X -118.2805,Y -76.4632,Z 183,A -143.3022,B 3.9405,C 0.2983,E1 3.8174,E2 236.3331} C_DIS
LIN {X -120.7704,Y -72.4673,Z 183,A -145.2649,B 3.9408,C 0.294,E1 3.8145,E2 238.3015} C_DIS
LIN {X -122.3932,Y -69.6904,Z 183,A -147.0083,B 3.9408,C 0.2937,E1 3.8121,E2 240.1016} C_DIS
LIN {X -124.5396,Y -65.7742,Z 183,A -148.3878,B 3.9414,C 0.2864,E1 3.8103,E2 241.4229} C_DIS
LIN {X -126.182,Y -62.5655,Z 183,A -149.8708,B 3.9416,C 0.2829,E1 3.8084,E2 242.9074} C_DIS
LIN {X -127.6935,Y -59.4201,Z 183,A -151.1409,B 3.9419,C 0.2784,E1 3.8069,E2 244.1571} C_DIS
LIN {X -129.5866,Y -55.1742,Z 183,A -153.4227,B 3.9421,C 0.276,E1 3.8043,E2 246.4897} C_DIS
LIN {X -131.0437,Y -51.6159,Z 183,A -154.951,B 3.9424,C 0.2717,E1 3.8027,E2 248.0126} C_DIS
LIN {X -134.0487,Y -43.2131,Z 183,A -158.7014,B 3.943,C 0.2628,E1 3.7993,E2 251.7769} C_DIS
LIN {X -135.1148,Y -39.7532,Z 183,A -160.1752,B 3.9433,C 0.2589,E1 3.7981,E2 253.25} C_DIS
LIN {X -136.062,Y -36.3791,Z 183,A -161.6644,B 3.9435,C 0.2554,E1 3.797,E2 254.7468} C_DIS
LIN {X -136.9026,Y -33.0758,Z 183,A -163.1016,B 3.9437,C 0.2519,E1 3.796,E2 256.1898} C_DIS
LIN {X -137.6409,Y -29.855,Z 183,A -164.5002,B 3.9439,C 0.2485,E1 3.7951,E2 257.5947} C_DIS
LIN {X -138.315,Y -26.5575,Z 183,A -166.6661,B 3.9439,C 0.2494,E1 3.794,E2 259.8632} C_DIS
LIN {X -139.2864,Y -20.8818,Z 183,A -168.4771,B 3.9445,C 0.2398,E1 3.7932,E2 261.6041} C_DIS
LIN {X -139.7466,Y -17.5451,Z 183,A -170.5967,B 3.9445,C 0.2403,E1 3.7925,E2 263.8198} C_DIS
LIN {X -140.3679,Y -11.5472,Z 183,A -172.2267,B 3.9451,C 0.2287,E1 3.7921,E2 265.3418} C_DIS
LIN {X -140.7277,Y -5.6694,Z 183,A -174.8306,B 3.9454,C 0.2231,E1 3.7917,E2 267.9712} C_DIS
LIN {X -140.8281,Y -1.996,Z 183,A -176.391,B 3.9457,C 0.2193,E1 3.7916,E2 269.5391} C_DIS
LIN {X -140.835,Y 1.5778,Z 183,A -178.1439,B 3.9457,C 0.2169,E1 3.7916,E2 271.3297} C_DIS
LIN {X -140.5265,Y 9.4517,Z 183,A 178.7084,B 3.9463,C 0.2075,E1 3.792,E2 274.4677} C_DIS
LIN {X -140.2133,Y 13.2907,Z 183,A 177.2364,B 3.9466,C 0.2025,E1 3.7924,E2 275.9261} C_DIS
LIN {X -139.7624,Y 17.4182,Z 183,A 174.5585,B 3.9466,C 0.2034,E1 3.7934,E2 278.7294} C_DIS
LIN {X -138.8441,Y 23.6408,Z 183,A 172.6414,B 3.9471,C 0.1926,E1 3.7942,E2 280.5628} C_DIS
LIN {X -138.2701,Y 26.7929,Z 183,A 171.1596,B 3.9471,C 0.19,E1 3.795,E2 282.0665} C_DIS
LIN {X -137.0584,Y 32.4293,Z 183,A 168.9343,B 3.9475,C 0.1829,E1 3.7963,E2 284.2747} C_DIS
LIN {X -136.1527,Y 36.039,Z 183,A 167.4488,B 3.9477,C 0.1786,E1 3.7973,E2 285.7553} C_DIS
LIN {X -135.3233,Y 39.0411,Z 183,A 166.027,B 3.9478,C 0.176,E1 3.7984,E2 287.1959} C_DIS
LIN {X -134.2522,Y 42.576,Z 183,A 164.4911,B 3.948,C 0.1721,E1 3.7997,E2 288.7348} C_DIS
LIN {X -133.1027,Y 46.0432,Z 183,A 163.0434,B 3.9482,C 0.1679,E1 3.801,E2 290.1765} C_DIS
LIN {X -132.0516,Y 48.9782,Z 183,A 161.6959,B 3.9482,C 0.165,E1 3.8023,E2 291.5331} C_DIS
LIN {X -130.7307,Y 52.4007,Z 183,A 160.1359,B 3.9484,C 0.1615,E1 3.8039,E2 293.1006} C_DIS
LIN {X -129.3939,Y 55.6199,Z 183,A 158.6878,B 3.9486,C 0.158,E1 3.8055,E2 294.5514} C_DIS
LIN {X -127.8767,Y 59.0237,Z 183,A 157.1484,B 3.9487,C 0.1543,E1 3.8072,E2 296.0925} C_DIS
LIN {X -126.3778,Y 62.1684,Z 183,A 155.6775,B 3.9489,C 0.151,E1 3.809,E2 297.5691} C_DIS
LIN {X -124.8277,Y 65.2255,Z 183,A 154.2115,B 3.9489,C 0.1479,E1 3.8109,E2 299.0431} C_DIS
LIN {X -122.4861,Y 69.5275,Z 183,A 152.0214,B 3.9491,C 0.1442,E1 3.8139,E2 301.2567} C_DIS
LIN {X -120.1563,Y 73.4801,Z 183,A 150.111,B 3.9493,C 0.14,E1 3.8167,E2 303.1711} C_DIS
LIN {X -117.7282,Y 77.3105,Z 183,A 148.4608,B 3.9495,C 0.1344,E1 3.8191,E2 304.7951} C_DIS
LIN {X -115.8914,Y 80.0379,Z 183,A 146.506,B 3.9495,C 0.1351,E1 3.8223,E2 306.8268} C_DIS
LIN {X -113.5465,Y 83.3307,Z 183,A 145.1582,B 3.9496,C 0.1296,E1 3.8245,E2 308.1359} C_DIS
LIN {X -110.8741,Y 86.855,Z 183,A 143.2916,B 3.9497,C 0.126,E1 3.8277,E2 310.0096} C_DIS
LIN {X -108.0111,Y 90.3906,Z 183,A 141.3848,B 3.9499,C 0.1224,E1 3.8311,E2 311.9219} C_DIS
LIN {X -105.052,Y 93.8133,Z 183,A 139.4879,B 3.9499,C 0.1189,E1 3.8346,E2 313.8245} C_DIS
LIN {X -101.9983,Y 97.1248,Z 183,A 137.5973,B 3.9501,C 0.1155,E1 3.8382,E2 315.7209} C_DIS
LIN {X -98.8159,Y 100.3609,Z 183,A 135.7164,B 3.9501,C 0.1121,E1 3.8419,E2 317.6047} C_DIS
LIN {X -95.5317,Y 103.492,Z 183,A 133.8057,B 3.9502,C 0.109,E1 3.8458,E2 319.522} C_DIS
LIN {X -92.1125,Y 106.5466,Z 183,A 131.9109,B 3.9503,C 0.1058,E1 3.8498,E2 321.4192} C_DIS
LIN {X -88.6886,Y 109.4133,Z 183,A 130.0308,B 3.9504,C 0.1031,E1 3.8539,E2 323.3057} C_DIS
LIN {X -85.0511,Y 112.264,Z 183,A 128.1237,B 3.9504,C 0.1001,E1 3.8581,E2 325.2149} C_DIS
LIN {X -81.3603,Y 114.9668,Z 183,A 126.2313,B 3.9505,C 0.0973,E1 3.8624,E2 327.1098} C_DIS
LIN {X -77.6223,Y 117.5229,Z 183,A 124.3674,B 3.9506,C 0.0947,E1 3.8667,E2 328.975} C_DIS
LIN {X -73.9122,Y 119.8912,Z 183,A 122.5038,B 3.9506,C 0.0926,E1 3.8711,E2 330.8465} C_DIS
LIN {X -69.9711,Y 122.233,Z 183,A 120.6197,B 3.9507,C 0.0902,E1 3.8757,E2 332.7317} C_DIS
LIN {X -66.0704,Y 124.3841,Z 183,A 118.8056,B 3.9507,C 0.0879,E1 3.8801,E2 334.5446} C_DIS
LIN {X -62.6701,Y 126.1304,Z 183,A 116.6226,B 3.9507,C 0.0906,E1 3.8858,E2 336.8045} C_DIS
LIN {X -57.7371,Y 128.463,Z 183,A 115.0631,B 3.9509,C 0.0833,E1 3.8895,E2 338.2806} C_DIS
LIN {X -51.7203,Y 131.0032,Z 183,A 112.0372,B 3.9509,C 0.0833,E1 3.8975,E2 341.3508} C_DIS
LIN {X -48.4367,Y 132.2523,Z 183,A 110.6245,B 3.9509,C 0.0819,E1 3.9012,E2 342.7605} C_DIS
LIN {X -45.2493,Y 133.377,Z 183,A 109.4,B 3.9509,C 0.0796,E1 3.9044,E2 343.9655} C_DIS
LIN {X -41.4568,Y 134.602,Z 183,A 107.9209,B 3.9509,C 0.0773,E1 3.9083,E2 345.4257} C_DIS
LIN {X -35.7073,Y 136.2412,Z 183,A 105.3096,B 3.9509,C 0.077,E1 3.9153,E2 348.058} C_DIS
LIN {X -31.4858,Y 137.277,Z 183,A 103.0573,B 3.9509,C 0.0799,E1 3.9216,E2 350.3693} C_DIS
LIN {X -26.576,Y 138.3115,Z 183,A 101.4935,B 3.951,C 0.0751,E1 3.9258,E2 351.8728} C_DIS
LIN {X -19.8593,Y 139.4345,Z 183,A 98.8053,B 3.951,C 0.0734,E1 3.9332,E2 354.5493} C_DIS
LIN {X -16.1759,Y 139.9106,Z 183,A 97.1781,B 3.951,C 0.074,E1 3.9377,E2 356.1903} C_DIS
LIN {X -12.159,Y 140.3162,Z 183,A 95.5769,B 3.951,C 0.0733,E1 3.9421,E2 357.7855} C_DIS
LIN {X -6.0888,Y 140.7114,Z 183,A 93.0723,B 3.951,C 0.0733,E1 3.9491,E2 360.2927} C_DIS
LIN {X -2.2393,Y 140.8241,Z 183,A 91.6034,B 3.951,C 0.0726,E1 3.9532,E2 361.7487} C_DIS
LIN {X 2.0192,Y 140.8277,Z 183,A 89.8439,B 3.951,C 0.073,E1 3.9581,E2 363.5109} C_DIS
LIN {X 5.6565,Y 140.7283,Z 183,A 88.3674,B 3.951,C 0.0732,E1 3.9622,E2 364.9863} C_DIS
LIN {X 10.1009,Y 140.4791,Z 183,A 86.6119,B 3.951,C 0.0732,E1 3.9671,E2 366.7342} C_DIS
LIN {X 13.4011,Y 140.2027,Z 183,A 85.3193,B 3.951,C 0.0732,E1 3.9707,E2 368.0194} C_DIS
LIN {X 16.5393,Y 139.8672,Z 183,A 83.9733,B 3.951,C 0.0742,E1 3.9745,E2 369.3727} C_DIS
LIN {X 19.6253,Y 139.4679,Z 183,A 82.4265,B 3.951,C 0.0774,E1 3.9788,E2 370.9541} C_DIS
LIN {X 22.9485,Y 138.9596,Z 183,A 81.4486,B 3.951,C 0.0745,E1 3.9814,E2 371.883} C_DIS
LIN {X 26.1035,Y 138.4018,Z 183,A 80.1032,B 3.951,C 0.0757,E1 3.9851,E2 373.2333} C_DIS
LIN {X 29.5019,Y 137.7172,Z 183,A 78.5957,B 3.951,C 0.0775,E1 3.9893,E2 374.7525} C_DIS
LIN {X 32.3715,Y 137.0724,Z 183,A 77.4906,B 3.951,C 0.0775,E1 3.9922,E2 375.846} C_DIS
LIN {X 36.5919,Y 136.0053,Z 183,A 75.6949,B 3.951,C 0.0791,E1 3.9971,E2 377.6443} C_DIS
LIN {X 39.7536,Y 135.1147,Z 183,A 73.9632,B 3.9508,C 0.0841,E1 4.0019,E2 379.425} C_DIS
LIN {X 43.8645,Y 133.8377,Z 183,A 72.5743,B 3.9508,C 0.0822,E1 4.0055,E2 380.7684} C_DIS
LIN {X 47.8667,Y 132.4578,Z 183,A 71.0035,B 3.9508,C 0.0825,E1 4.0095,E2 382.3199} C_DIS
LIN {X 50.7944,Y 131.3631,Z 183,A 69.8149,B 3.9508,C 0.083,E1 4.0126,E2 383.4979} C_DIS
LIN {X 53.7905,Y 130.1658,Z 183,A 68.4114,B 3.9508,C 0.0854,E1 4.0163,E2 384.9126} C_DIS
LIN {X 57.3676,Y 128.6283,Z 183,A 66.9196,B 3.9508,C 0.0864,E1 4.0201,E2 386.3926} C_DIS
LIN {X 60.3779,Y 127.2434,Z 183,A 65.5383,B 3.9508,C 0.0884,E1 4.0236,E2 387.778} C_DIS
LIN {X 65.9346,Y 124.4553,Z 183,A 63.0356,B 3.9507,C 0.0916,E1 4.0298,E2 390.2772} C_DIS
LIN {X 69.7912,Y 122.3356,Z 183,A 61.2584,B 3.9507,C 0.094,E1 4.0341,E2 392.0527} C_DIS
LIN {X 73.3874,Y 120.2132,Z 183,A 59.5363,B 3.9506,C 0.0968,E1 4.0383,E2 393.7777} C_DIS
LIN {X 77.1335,Y 117.8448,Z 183,A 57.7521,B 3.9505,C 0.0995,E1 4.0425,E2 395.5596} C_DIS
LIN {X 80.1388,Y 115.8219,Z 183,A 56.041,B 3.9504,C 0.1045,E1 4.0465,E2 397.3005} C_DIS
LIN {X 83.2958,Y 113.5722,Z 183,A 54.7901,B 3.9504,C 0.1037,E1 4.0492,E2 398.5105} C_DIS
LIN {X 86.9746,Y 110.7801,Z 183,A 52.9539,B 3.9504,C 0.1066,E1 4.0532,E2 400.3415} C_DIS
LIN {X 90.4767,Y 107.9388,Z 183,A 51.1654,B 3.9502,C 0.1095,E1 4.0571,E2 402.1244} C_DIS
LIN {X 93.3714,Y 105.4448,Z 183,A 49.4198,B 3.9501,C 0.1145,E1 4.0608,E2 403.8943} C_DIS
LIN {X 95.9593,Y 103.0948,Z 183,A 47.8374,B 3.95,C 0.119,E1 4.0641,E2 405.4971} C_DIS
LIN {X 99.3158,Y 99.8659,Z 183,A 46.4297,B 3.95,C 0.1175,E1 4.0668,E2 406.8436} C_DIS
LIN {X 102.4816,Y 96.6144,Z 183,A 44.6573,B 3.95,C 0.1206,E1 4.0702,E2 408.607} C_DIS
LIN {X 105.2186,Y 93.627,Z 183,A 42.9835,B 3.9498,C 0.1244,E1 4.0733,E2 410.2844} C_DIS
LIN {X 108.1578,Y 90.215,Z 183,A 40.7033,B 3.9495,C 0.1334,E1 4.0775,E2 412.6218} C_DIS
LIN {X 111.4338,Y 86.1356,Z 183,A 39.1613,B 3.9495,C 0.1316,E1 4.08,E2 414.09} C_DIS
LIN {X 114.1718,Y 82.4722,Z 183,A 37.3542,B 3.9495,C 0.1353,E1 4.083,E2 415.8908} C_DIS
LIN {X 116.8345,Y 78.6553,Z 183,A 35.5336,B 3.9493,C 0.1389,E1 4.0859,E2 417.7028} C_DIS
LIN {X 119.2207,Y 74.9887,Z 183,A 33.7855,B 3.9492,C 0.1428,E1 4.0885,E2 419.4475} C_DIS
LIN {X 121.637,Y 71.0029,Z 183,A 31.9342,B 3.949,C 0.1469,E1 4.0911,E2 421.2938} C_DIS
LIN {X 123.842,Y 67.0831,Z 183,A 30.1713,B 3.9489,C 0.1507,E1 4.0935,E2 423.0488} C_DIS
LIN {X 125.4566,Y 64.007,Z 183,A 28.898,B 3.9488,C 0.1526,E1 4.0951,E2 424.3046} C_DIS
LIN {X 126.9846,Y 60.9197,Z 183,A 27.5421,B 3.9487,C 0.1557,E1 4.0968,E2 425.6552} C_DIS
LIN {X 128.4502,Y 57.7659,Z 183,A 26.2023,B 3.9486,C 0.1584,E1 4.0983,E2 426.986} C_DIS
LIN {X 129.8946,Y 54.4398,Z 183,A 24.722,B 3.9484,C 0.1623,E1 4.0999,E2 428.4677} C_DIS
LIN {X 131.1984,Y 51.2182,Z 183,A 23.4209,B 3.9484,C 0.1647,E1 4.1013,E2 429.7549} C_DIS
LIN {X 132.3618,Y 48.1329,Z 183,A 22.0349,B 3.9481,C 0.1688,E1 4.1026,E2 431.1473} C_DIS
LIN {X 133.4672,Y 44.9785,Z 183,A 20.7412,B 3.9481,C 0.1717,E1 4.1038,E2 432.4332} C_DIS
LIN {X 134.6041,Y 41.45,Z 183,A 19.3071,B 3.9479,C 0.1749,E1 4.105,E2 433.8584} C_DIS
LIN {X 136.5795,Y 34.3864,Z 183,A 15.9286,B 3.9473,C 0.1878,E1 4.1075,E2 437.2896} C_DIS
LIN {X 137.6217,Y 29.9442,Z 183,A 14.2289,B 3.9471,C 0.191,E1 4.1085,E2 438.9701} C_DIS
LIN {X 138.4321,Y 25.9454,Z 183,A 12.672,B 3.947,C 0.1944,E1 4.1093,E2 440.5148} C_DIS
LIN {X 139.0837,Y 22.1924,Z 183,A 11.4043,B 3.947,C 0.1953,E1 4.1098,E2 441.7469} C_DIS
LIN {X 139.6197,Y 18.5137,Z 183,A 10.1215,B 3.9468,C 0.1968,E1 4.1103,E2 443.0008} C_DIS
LIN {X 140.1849,Y 13.5862,Z 183,A 8.0858,B 3.9465,C 0.2027,E1 4.1109,E2 445.0401} C_DIS
LIN {X 140.5139,Y 9.6248,Z 183,A 6.4892,B 3.9463,C 0.207,E1 4.1113,E2 446.6351} C_DIS
LIN {X 140.7285,Y 5.6505,Z 183,A 4.9989,B 3.9462,C 0.21,E1 4.1115,E2 448.1097} C_DIS
LIN {X 140.8234,Y 2.2782,Z 183,A 3.6093,B 3.9459,C 0.2141,E1 4.1115,E2 449.5024} C_DIS
LIN {X 140.8299,Y -1.8862,Z 183,A 2.0438,B 3.9458,C 0.2173,E1 4.1115,E2 451.0523} C_DIS
LIN {X 140.7365,Y -5.4456,Z 183,A 0.6589,B 3.9456,C 0.2207,E1 4.1115,E2 452.4298} C_DIS
LIN {X 140.5568,Y -8.959,Z 183,A -0.8329,B 3.9453,C 0.2255,E1 4.1112,E2 453.9306} C_DIS
LIN {X 140.2149,Y -13.2744,Z 183,A -2.449,B 3.9451,C 0.2287,E1 4.1108,E2 455.529} C_DIS
LIN {X 139.8424,Y -16.7472,Z 183,A -3.8709,B 3.9449,C 0.2327,E1 4.1103,E2 456.9521} C_DIS
LIN {X 139.1659,Y -21.6616,Z 183,A -5.79,B 3.9446,C 0.2371,E1 4.1096,E2 458.8596} C_DIS
LIN {X 138.4634,Y -25.7815,Z 183,A -7.3374,B 3.9445,C 0.24,E1 4.1088,E2 460.3882} C_DIS
LIN {X 137.4711,Y -30.6361,Z 183,A -9.4299,B 3.9441,C 0.2466,E1 4.1076,E2 462.4925} C_DIS
LIN {X 136.5266,Y -34.5948,Z 183,A -11.3035,B 3.9436,C 0.2538,E1 4.1063,E2 464.3961} C_DIS
LIN {X 135.5401,Y -38.2794,Z 183,A -12.478,B 3.9436,C 0.2535,E1 4.1055,E2 465.522} C_DIS
LIN {X 133.8301,Y -43.8887,Z 183,A -14.6756,B 3.9433,C 0.2577,E1 4.1037,E2 467.6966} C_DIS
LIN {X 132.4293,Y -47.9457,Z 183,A -16.5723,B 3.9429,C 0.2642,E1 4.1019,E2 469.6148} C_DIS
LIN {X 130.7758,Y -52.2889,Z 183,A -18.321,B 3.9427,C 0.2675,E1 4.1002,E2 471.3462} C_DIS
LIN {X 129.3712,Y -55.6724,Z 183,A -19.6878,B 3.9425,C 0.27,E1 4.0987,E2 472.6978} C_DIS
LIN {X 126.3943,Y -62.135,Z 183,A -23.2371,B 3.9414,C 0.2853,E1 4.0943,E2 476.3361} C_DIS
LIN {X 123.6359,Y -67.461,Z 183,A -24.7508,B 3.9418,C 0.2805,E1 4.0925,E2 477.7291} C_DIS
LIN {X 120.55,Y -72.8321,Z 183,A -27.3946,B 3.9412,C 0.2882,E1 4.0888,E2 480.3916} C_DIS
LIN {X 118.2228,Y -76.5521,Z 183,A -29.1513,B 3.9409,C 0.2922,E1 4.0861,E2 482.146} C_DIS
LIN {X 115.6179,Y -80.4321,Z 183,A -30.9808,B 3.9407,C 0.2959,E1 4.0832,E2 483.9676} C_DIS
LIN {X 112.9303,Y -84.164,Z 183,A -32.7776,B 3.9404,C 0.2994,E1 4.0803,E2 485.756} C_DIS
LIN {X 110.1757,Y -87.739,Z 183,A -34.5831,B 3.9401,C 0.3033,E1 4.0772,E2 487.559} C_DIS
LIN {X 107.154,Y -91.4052,Z 183,A -36.4326,B 3.9398,C 0.3066,E1 4.0739,E2 489.399} C_DIS
LIN {X 104.3311,Y -94.6141,Z 183,A -38.4712,B 3.9393,C 0.3139,E1 4.07,E2 491.4791} C_DIS
LIN {X 101.532,Y -97.6127,Z 183,A -40.4144,B 3.9387,C 0.3205,E1 4.0662,E2 493.4603} C_DIS
LIN {X 97.3817,Y -101.7528,Z 183,A -41.8883,B 3.9392,C 0.315,E1 4.0635,E2 494.8143} C_DIS
LIN {X 92.2282,Y -106.4469,Z 183,A -45.5585,B 3.938,C 0.33,E1 4.0556,E2 498.5986} C_DIS
LIN {X 87.4694,Y -110.3903,Z 183,A -47.1986,B 3.9384,C 0.3249,E1 4.0522,E2 500.1237} C_DIS
LIN {X 81.2658,Y -115.0335,Z 183,A -50.8469,B 3.9375,C 0.336,E1 4.0439,E2 503.8413} C_DIS
LIN {X 77.3323,Y -117.7139,Z 183,A -52.2846,B 3.9376,C 0.3337,E1 4.0407,E2 505.2135} C_DIS
LIN {X 73.4492,Y -120.1753,Z 183,A -54.0243,B 3.9376,C 0.3353,E1 4.0366,E2 506.937} C_DIS
LIN {X 71.2161,Y -121.5117,Z 183,A -55.1572,B 3.9373,C 0.3377,E1 4.0338,E2 508.0807} C_DIS
LIN {X 68.0023,Y -123.3393,Z 183,A -56.6715,B 3.9371,C 0.3401,E1 4.0301,E2 509.5976} C_DIS
LIN {X 64.1851,Y -125.3659,Z 183,A -58.2994,B 3.9371,C 0.3412,E1 4.0261,E2 511.2091} C_DIS
LIN {X 60.937,Y -126.9764,Z 183,A -59.7483,B 3.9369,C 0.3429,E1 4.0225,E2 512.6556} C_DIS
LIN {X 57.7075,Y -128.4763,Z 183,A -61.0973,B 3.9368,C 0.3437,E1 4.0191,E2 513.9921} C_DIS
LIN {X 54.5203,Y -129.861,Z 183,A -62.4562,B 3.9367,C 0.3449,E1 4.0156,E2 515.3447} C_DIS
LIN {X 51.7166,Y -131.0046,Z 183,A -63.8697,B 3.9364,C 0.3483,E1 4.0119,E2 516.7837} C_DIS
LIN {X 48.2407,Y -132.323,Z 183,A -65.745,B 3.9359,C 0.3537,E1 4.0069,E2 518.7089} C_DIS
LIN {X 43.982,Y -133.799,Z 183,A -67.1185,B 3.9362,C 0.3508,E1 4.0034,E2 520.0216} C_DIS
LIN {X 40.0488,Y -135.0283,Z 183,A -68.7743,B 3.936,C 0.3522,E1 3.9989,E2 521.6758} C_DIS
LIN {X 36.2254,Y -136.103,Z 183,A -70.3385,B 3.936,C 0.3531,E1 3.9947,E2 523.234} C_DIS
LIN {X 32.4311,Y -137.058,Z 183,A -71.9397,B 3.9358,C 0.3545,E1 3.9904,E2 524.8375} C_DIS
LIN {X 28.4748,Y -137.9336,Z 183,A -73.5894,B 3.9358,C 0.3557,E1 3.9859,E2 526.4884} C_DIS
LIN {X 24.3525,Y -138.721,Z 183,A -75.3584,B 3.9356,C 0.3574,E1 3.981,E2 528.2667} C_DIS
LIN {X 17.4728,Y -139.7559,Z 183,A -78.1431,B 3.9355,C 0.3585,E1 3.9733,E2 531.0469} C_DIS
LIN {X 13.3959,Y -140.2032,Z 183,A -79.7342,B 3.9355,C 0.3585,E1 3.9689,E2 532.6284} C_DIS
LIN {X 9.1665,Y -140.544,Z 183,A -81.4671,B 3.9355,C 0.3591,E1 3.9641,E2 534.3632} C_DIS
LIN {X 5.6149,Y -140.7299,Z 183,A -82.8727,B 3.9355,C 0.3591,E1 3.9602,E2 535.7638} C_DIS
LIN {X 1.6797,Y -140.8334,Z 183,A -84.5179,B 3.9353,C 0.3599,E1 3.9555,E2 537.4159} C_DIS
LIN {X 1.6797,Y -140.8334,Z 183,A -84.5179,B 3.9353,C 0.3599,E1 3.9555,E2 537.4159} C_DIS
Enddeposition()
LIN {X 0.9913,Y -141.7363,Z 183,A -84.3151,B 3.9358,C 0.3575,E1 3.9564,E2 537.1786} C_DIS
Startdeposition()
$VEL.CP = VEL_PRINT
LIN {X 3.9067,Y -141.689,Z 183,A -82.8965,B 3.936,C 0.3549,E1 3.9605,E2 535.7265} C_DIS
LIN {X 7.5732,Y -141.5411,Z 183,A -81.3174,B 3.9361,C 0.3536,E1 3.9649,E2 534.1334} C_DIS
LIN {X 11.3883,Y -141.2855,Z 183,A -79.8144,B 3.9361,C 0.3535,E1 3.9691,E2 532.6356} C_DIS
LIN {X 15.129,Y -140.933,Z 183,A -78.3125,B 3.9361,C 0.353,E1 3.9732,E2 531.1351} C_DIS
LIN {X 20.1862,Y -140.2979,Z 183,A -76.2262,B 3.9363,C 0.3516,E1 3.979,E2 529.044} C_DIS
LIN {X 24.7977,Y -139.5567,Z 183,A -74.4446,B 3.9363,C 0.3516,E1 3.9839,E2 527.2761} C_DIS
LIN {X 28.0574,Y -138.938,Z 183,A -73.1273,B 3.9363,C 0.3509,E1 3.9875,E2 525.9613} C_DIS
LIN {X 31.4718,Y -138.2045,Z 183,A -71.6945,B 3.9365,C 0.3496,E1 3.9914,E2 524.5247} C_DIS
LIN {X 35.3564,Y -137.2629,Z 183,A -70.1318,B 3.9365,C 0.3488,E1 3.9957,E2 522.9682} C_DIS
LIN {X 38.4215,Y -136.436,Z 183,A -68.7903,B 3.9367,C 0.3471,E1 3.9993,E2 521.6179} C_DIS
LIN {X 42.8371,Y -135.1147,Z 183,A -67.1348,B 3.9367,C 0.3475,E1 4.0036,E2 519.9899} C_DIS
LIN {X 46.6828,Y -133.8346,Z 183,A -65.3925,B 3.9369,C 0.3447,E1 4.0083,E2 518.2321} C_DIS
LIN {X 50.7066,Y -132.364,Z 183,A -63.5851,B 3.9371,C 0.3419,E1 4.0131,E2 516.4132} C_DIS
LIN {X 53.8044,Y -131.1361,Z 183,A -62.2577,B 3.9373,C 0.3406,E1 4.0165,E2 515.0875} C_DIS
LIN {X 57.3267,Y -129.6336,Z 183,A -60.8421,B 3.9373,C 0.3401,E1 4.0201,E2 513.6891} C_DIS
LIN {X 60.5871,Y -128.1421,Z 183,A -59.3661,B 3.9375,C 0.3379,E1 4.0238,E2 512.2082} C_DIS
LIN {X 63.7912,Y -126.5775,Z 183,A -57.9353,B 3.9376,C 0.336,E1 4.0274,E2 510.7779} C_DIS
LIN {X 67.0459,Y -124.8851,Z 183,A -56.1788,B 3.9381,C 0.3308,E1 4.0318,E2 508.9825} C_DIS
LIN {X 70.4429,Y -123.001,Z 183,A -54.9496,B 3.938,C 0.3323,E1 4.0347,E2 507.7993} C_DIS
LIN {X 73.8154,Y -121.0073,Z 183,A -53.2946,B 3.9382,C 0.329,E1 4.0387,E2 506.1332} C_DIS
LIN {X 77.6278,Y -118.5981,Z 183,A -50.935,B 3.939,C 0.3199,E1 4.0444,E2 503.6979} C_DIS
LIN {X 82.5561,Y -115.2213,Z 183,A -49.2592,B 3.9386,C 0.3241,E1 4.048,E2 502.1225} C_DIS
LIN {X 85.9712,Y -112.6961,Z 183,A -47.5377,B 3.9389,C 0.321,E1 4.0518,E2 500.399} C_DIS
LIN {X 88.4984,Y -110.7229,Z 183,A -45.986,B 3.9393,C 0.3157,E1 4.0553,E2 498.811} C_DIS
LIN {X 91.5196,Y -108.2387,Z 183,A -44.5406,B 3.9394,C 0.3142,E1 4.0583,E2 497.3831} C_DIS
LIN {X 94.0751,Y -106.0254,Z 183,A -43.3923,B 3.9394,C 0.3141,E1 4.0607,E2 496.2637} C_DIS
LIN {X 97.4402,Y -102.9412,Z 183,A -41.7046,B 3.9396,C 0.3122,E1 4.0641,E2 494.596} C_DIS
LIN {X 102.0199,Y -98.4045,Z 183,A -38.9127,B 3.9402,C 0.3046,E1 4.0696,E2 491.7765} C_DIS
LIN {X 106.6179,Y -93.403,Z 183,A -36.5088,B 3.9403,C 0.3027,E1 4.0741,E2 489.4173} C_DIS
LIN {X 109.5618,Y -89.9319,Z 183,A -34.5729,B 3.9407,C 0.2974,E1 4.0775,E2 487.4667} C_DIS
LIN {X 112.4571,Y -86.2838,Z 183,A -32.7831,B 3.941,C 0.2942,E1 4.0806,E2 485.688} C_DIS
LIN {X 115.0523,Y -82.7925,Z 183,A -31.0642,B 3.9413,C 0.2906,E1 4.0834,E2 483.9731} C_DIS
LIN {X 117.6557,Y -79.0491,Z 183,A -29.2786,B 3.9415,C 0.2869,E1 4.0862,E2 482.1938} C_DIS
LIN {X 120.0695,Y -75.332,Z 183,A -27.5224,B 3.9418,C 0.2829,E1 4.0889,E2 480.4409} C_DIS
LIN {X 122.7418,Y -70.8937,Z 183,A -25.3385,B 3.9423,C 0.2766,E1 4.092,E2 478.2429} C_DIS
LIN {X 124.3332,Y -68.0643,Z 183,A -24.2814,B 3.9423,C 0.2764,E1 4.0934,E2 477.2195} C_DIS
LIN {X 126.1154,Y -64.699,Z 183,A -22.8265,B 3.9425,C 0.2735,E1 4.0952,E2 475.7747} C_DIS
LIN {X 127.683,Y -61.5481,Z 183,A -21.5843,B 3.9425,C 0.2721,E1 4.0967,E2 474.5558} C_DIS
LIN {X 129.4716,Y -57.6891,Z 183,A -19.8021,B 3.9429,C 0.2668,E1 4.0988,E2 472.7637} C_DIS
LIN {X 130.7722,Y -54.6764,Z 183,A -18.5551,B 3.9431,C 0.2643,E1 4.1001,E2 471.5264} C_DIS
LIN {X 131.9351,Y -51.8098,Z 183,A -17.2398,B 3.9434,C 0.2602,E1 4.1015,E2 470.2013} C_DIS
LIN {X 134.2922,Y -45.3528,Z 183,A -14.7044,B 3.9437,C 0.2557,E1 4.1039,E2 467.6966} C_DIS
LIN {X 136.3963,Y -38.5634,Z 183,A -11.5263,B 3.9444,C 0.2441,E1 4.1065,E2 464.4751} C_DIS
LIN {X 137.3132,Y -35.1584,Z 183,A -10.4361,B 3.9444,C 0.2443,E1 4.1072,E2 463.429} C_DIS
LIN {X 138.1677,Y -31.6326,Z 183,A -9.0736,B 3.9446,C 0.2416,E1 4.1081,E2 462.0794} C_DIS
LIN {X 139.0341,Y -27.5855,Z 183,A -7.3447,B 3.9449,C 0.2362,E1 4.109,E2 460.3417} C_DIS
LIN {X 139.7551,Y -23.6556,Z 183,A -5.7954,B 3.9451,C 0.2325,E1 4.1098,E2 458.8} C_DIS
LIN {X 140.2898,Y -20.2431,Z 183,A -4.5077,B 3.9452,C 0.2299,E1 4.1103,E2 457.5258} C_DIS
LIN {X 140.7103,Y -17.0791,Z 183,A -3.2027,B 3.9455,C 0.2261,E1 4.1108,E2 456.2179} C_DIS
LIN {X 141.1236,Y -13.2376,Z 183,A -1.7489,B 3.9456,C 0.2231,E1 4.1112,E2 454.7775} C_DIS
LIN {X 141.4532,Y -9.062,Z 183,A -0.1279,B 3.9459,C 0.2192,E1 4.1115,E2 453.1649} C_DIS
LIN {X 141.6455,Y -5.2574,Z 183,A 1.1958,B 3.9459,C 0.2175,E1 4.1117,E2 451.869} C_DIS
LIN {X 141.7261,Y -2.1849,Z 183,A 2.616,B 3.9463,C 0.2118,E1 4.1117,E2 450.4241} C_DIS
LIN {X 141.7252,Y 2.239,Z 183,A 4.3302,B 3.9465,C 0.2076,E1 4.1117,E2 448.7186} C_DIS
LIN {X 141.5841,Y 6.7165,Z 183,A 5.9803,B 3.9466,C 0.2045,E1 4.1115,E2 447.0887} C_DIS
LIN {X 141.3955,Y 9.9232,Z 183,A 7.2997,B 3.9468,C 0.2006,E1 4.1113,E2 445.7656} C_DIS
LIN {X 141.1031,Y 13.4507,Z 183,A 8.7692,B 3.9471,C 0.196,E1 4.1109,E2 444.2901} C_DIS
LIN {X 140.5661,Y 18.226,Z 183,A 10.5369,B 3.9472,C 0.1927,E1 4.1103,E2 442.5444} C_DIS
LIN {X 140.1325,Y 21.3073,Z 183,A 11.8429,B 3.9474,C 0.1886,E1 4.1098,E2 441.2312} C_DIS
LIN {X 139.4903,Y 25.1685,Z 183,A 13.6164,B 3.9478,C 0.1819,E1 4.1089,E2 439.4313} C_DIS
LIN {X 138.7662,Y 28.9017,Z 183,A 14.8401,B 3.9478,C 0.1815,E1 4.1083,E2 438.2484} C_DIS
LIN {X 137.8873,Y 32.8358,Z 183,A 16.3454,B 3.9479,C 0.1785,E1 4.1073,E2 436.7587} C_DIS
LIN {X 137.0324,Y 36.237,Z 183,A 17.7356,B 3.9481,C 0.1749,E1 4.1063,E2 435.3712} C_DIS
LIN {X 135.7674,Y 40.7276,Z 183,A 19.6388,B 3.9483,C 0.1696,E1 4.1049,E2 433.4648} C_DIS
LIN {X 134.5158,Y 44.6812,Z 183,A 21.1668,B 3.9484,C 0.1669,E1 4.1036,E2 431.9554} C_DIS
LIN {X 133.333,Y 48.0959,Z 183,A 22.5327,B 3.9485,C 0.1641,E1 4.1023,E2 430.6014} C_DIS
LIN {X 132.1083,Y 51.3643,Z 183,A 23.9502,B 3.9487,C 0.1603,E1 4.1009,E2 429.1822} C_DIS
LIN {X 130.6355,Y 55.0038,Z 183,A 25.5209,B 3.9488,C 0.1563,E1 4.0992,E2 427.613} C_DIS
LIN {X 128.8334,Y 59.1017,Z 183,A 27.2513,B 3.949,C 0.1526,E1 4.0972,E2 425.8922} C_DIS
LIN {X 127.2571,Y 62.4227,Z 183,A 28.5817,B 3.949,C 0.1506,E1 4.0957,E2 424.5815} C_DIS
LIN {X 125.6979,Y 65.5063,Z 183,A 30.0426,B 3.9492,C 0.1463,E1 4.0938,E2 423.1117} C_DIS
LIN {X 123.5445,Y 69.4852,Z 183,A 31.8549,B 3.9494,C 0.142,E1 4.0913,E2 421.3009} C_DIS
LIN {X 121.3154,Y 73.3077,Z 183,A 33.5797,B 3.9495,C 0.1383,E1 4.0889,E2 419.5838} C_DIS
LIN {X 119.0231,Y 76.974,Z 183,A 35.3186,B 3.9497,C 0.1342,E1 4.0863,E2 417.8455} C_DIS
LIN {X 116.418,Y 80.8598,Z 183,A 37.1246,B 3.9497,C 0.1308,E1 4.0835,E2 416.05} C_DIS
LIN {X 113.9117,Y 84.3546,Z 183,A 38.8394,B 3.9499,C 0.127,E1 4.0806,E2 414.3377} C_DIS
LIN {X 109.2849,Y 90.2679,Z 183,A 41.7796,B 3.9501,C 0.1213,E1 4.0755,E2 411.4091} C_DIS
LIN {X 106.4744,Y 93.5672,Z 183,A 43.5521,B 3.9501,C 0.1173,E1 4.0723,E2 409.6336} C_DIS
LIN {X 103.1273,Y 97.243,Z 183,A 45.4429,B 3.9503,C 0.1144,E1 4.0687,E2 407.7579} C_DIS
LIN {X 99.8076,Y 100.6474,Z 183,A 48.3021,B 3.9507,C 0.1,E1 4.0628,E2 404.7757} C_DIS
LIN {X 93.9914,Y 106.0994,Z 183,A 50.3519,B 3.9505,C 0.1068,E1 4.0589,E2 402.8788} C_DIS
LIN {X 90.0223,Y 109.4879,Z 183,A 52.5467,B 3.9506,C 0.102,E1 4.0542,E2 400.6728} C_DIS
LIN {X 86.4828,Y 112.3047,Z 183,A 54.3346,B 3.9506,C 0.0991,E1 4.0502,E2 398.89} C_DIS
LIN {X 83.7866,Y 114.3296,Z 183,A 55.6698,B 3.9507,C 0.0971,E1 4.0472,E2 397.5584} C_DIS
LIN {X 79.8273,Y 117.1289,Z 183,A 57.5803,B 3.9508,C 0.0944,E1 4.0429,E2 395.6542} C_DIS
LIN {X 76.0463,Y 119.6186,Z 183,A 59.3736,B 3.9508,C 0.0918,E1 4.0387,E2 393.8656} C_DIS
LIN {X 72.3081,Y 121.9142,Z 183,A 61.0919,B 3.9509,C 0.0897,E1 4.0346,E2 392.1545} C_DIS
LIN {X 68.275,Y 124.2182,Z 183,A 62.9016,B 3.9509,C 0.0877,E1 4.0302,E2 390.3535} C_DIS
LIN {X 64.7938,Y 126.0671,Z 183,A 64.3897,B 3.9509,C 0.0866,E1 4.0265,E2 388.879} C_DIS
LIN {X 61.6466,Y 127.6359,Z 183,A 65.8804,B 3.951,C 0.0841,E1 4.0228,E2 387.3796} C_DIS
LIN {X 58.0635,Y 129.3041,Z 183,A 67.4494,B 3.951,C 0.0824,E1 4.0188,E2 385.8144} C_DIS
LIN {X 54.8486,Y 130.7003,Z 183,A 68.7819,B 3.951,C 0.0816,E1 4.0154,E2 384.4929} C_DIS
LIN {X 51.3923,Y 132.0974,Z 183,A 70.2692,B 3.9511,C 0.0801,E1 4.0115,E2 383.0083} C_DIS
LIN {X 48.3106,Y 133.2556,Z 183,A 72.0357,B 3.9512,C 0.0743,E1 4.0068,E2 381.186} C_DIS
LIN {X 44.1087,Y 134.7059,Z 183,A 73.977,B 3.9512,C 0.0712,E1 4.0015,E2 379.2265} C_DIS
LIN {X 38.966,Y 136.2837,Z 183,A 75.6008,B 3.9512,C 0.0747,E1 3.9974,E2 377.6741} C_DIS
LIN {X 34.0199,Y 137.6017,Z 183,A 77.6536,B 3.9512,C 0.0733,E1 3.9918,E2 375.624} C_DIS
LIN {X 30.6104,Y 138.3996,Z 183,A 78.9948,B 3.9512,C 0.073,E1 3.9882,E2 374.2926} C_DIS
LIN {X 27.48,Y 139.0555,Z 183,A 80.3197,B 3.9512,C 0.0719,E1 3.9846,E2 372.964} C_DIS
LIN {X 23.6728,Y 139.7522,Z 183,A 81.7288,B 3.9512,C 0.0725,E1 3.9807,E2 371.5752} C_DIS
LIN {X 19.968,Y 140.3291,Z 183,A 83.2913,B 3.9512,C 0.0713,E1 3.9764,E2 370.0072} C_DIS
LIN {X 16.1075,Y 140.8262,Z 183,A 84.9314,B 3.9513,C 0.07,E1 3.9718,E2 368.3592} C_DIS
LIN {X 11.8832,Y 141.2437,Z 183,A 86.5421,B 3.9513,C 0.0704,E1 3.9674,E2 366.7625} C_DIS
LIN {X 7.9456,Y 141.522,Z 183,A 88.2644,B 3.9513,C 0.0688,E1 3.9625,E2 365.0247} C_DIS
LIN {X 3.6271,Y 141.6968,Z 183,A 89.9947,B 3.9513,C 0.0686,E1 3.9577,E2 363.2972} C_DIS
LIN {X -0.5872,Y 141.7418,Z 183,A 91.5892,B 3.9513,C 0.0694,E1 3.9533,E2 361.7174} C_DIS
LIN {X -4.3144,Y 141.6777,Z 183,A 93.2004,B 3.9513,C 0.0685,E1 3.9488,E2 360.0935} C_DIS
LIN {X -8.5024,Y 141.4877,Z 183,A 94.7743,B 3.9513,C 0.0697,E1 3.9444,E2 358.5358} C_DIS
LIN {X -11.7774,Y 141.2527,Z 183,A 96.232,B 3.9513,C 0.0687,E1 3.9403,E2 357.0621} C_DIS
LIN {X -16.4225,Y 140.7886,Z 183,A 97.9062,B 3.9513,C 0.071,E1 3.9357,E2 355.4159} C_DIS
LIN {X -19.8588,Y 140.3447,Z 183,A 99.5707,B 3.9513,C 0.0691,E1 3.931,E2 353.7186} C_DIS
LIN {X -27.0993,Y 139.1288,Z 183,A 102.4579,B 3.9513,C 0.0711,E1 3.9231,E2 350.8434} C_DIS
LIN {X -31.2068,Y 138.265,Z 183,A 104.1,B 3.9513,C 0.0724,E1 3.9187,E2 349.2091} C_DIS
LIN {X -34.4419,Y 137.495,Z 183,A 105.3176,B 3.9513,C 0.0742,E1 3.9154,E2 348.0085} C_DIS
LIN {X -39.2791,Y 136.1925,Z 183,A 107.5734,B 3.9513,C 0.0737,E1 3.9093,E2 345.7245} C_DIS
LIN {X -42.5758,Y 135.1982,Z 183,A 108.9858,B 3.9513,C 0.0746,E1 3.9055,E2 344.3104} C_DIS
LIN {X -46.1309,Y 134.0259,Z 183,A 111.0253,B 3.9513,C 0.0717,E1 3.8999,E2 342.2044} C_DIS
LIN {X -50.7895,Y 132.3317,Z 183,A 112.4063,B 3.9512,C 0.0785,E1 3.8965,E2 340.9044} C_DIS
LIN {X -53.9144,Y 131.0905,Z 183,A 113.9536,B 3.9512,C 0.0783,E1 3.8924,E2 339.3341} C_DIS
LIN {X -57.639,Y 129.494,Z 183,A 115.4933,B 3.9512,C 0.0808,E1 3.8885,E2 337.808} C_DIS
LIN {X -62.5639,Y 127.1874,Z 183,A 117.771,B 3.9511,C 0.0828,E1 3.8828,E2 335.5217} C_DIS
LIN {X -65.7459,Y 125.5722,Z 183,A 119.1935,B 3.9511,C 0.0847,E1 3.8792,E2 334.1027} C_DIS
LIN {X -69.5203,Y 123.5248,Z 183,A 121.0513,B 3.951,C 0.0861,E1 3.8747,E2 332.2307} C_DIS
LIN {X -73.4568,Y 121.2252,Z 183,A 122.9633,B 3.951,C 0.0881,E1 3.87,E2 330.3111} C_DIS
LIN {X -77.4459,Y 118.7168,Z 183,A 124.9036,B 3.9509,C 0.0907,E1 3.8655,E2 328.3677} C_DIS
LIN {X -81.2912,Y 116.1178,Z 183,A 126.8398,B 3.9509,C 0.0931,E1 3.861,E2 326.4251} C_DIS
LIN {X -85.0746,Y 113.375,Z 183,A 128.7595,B 3.9508,C 0.096,E1 3.8567,E2 324.503} C_DIS
LIN {X -88.6705,Y 110.5855,Z 183,A 130.6035,B 3.9507,C 0.0991,E1 3.8526,E2 322.6597} C_DIS
LIN {X -92.1054,Y 107.7413,Z 183,A 132.4783,B 3.9507,C 0.1018,E1 3.8486,E2 320.7771} C_DIS
LIN {X -95.5845,Y 104.6673,Z 183,A 134.4223,B 3.9505,C 0.1048,E1 3.8446,E2 318.826} C_DIS
LIN {X -98.9527,Y 101.4888,Z 183,A 136.3351,B 3.9505,C 0.1082,E1 3.8407,E2 316.9093} C_DIS
LIN {X -102.1615,Y 98.2582,Z 183,A 138.1947,B 3.9504,C 0.1117,E1 3.8371,E2 315.0487} C_DIS
LIN {X -105.2444,Y 94.9485,Z 183,A 140.0943,B 3.9503,C 0.115,E1 3.8335,E2 313.1415} C_DIS
LIN {X -108.1306,Y 91.6475,Z 183,A 141.8907,B 3.9502,C 0.1186,E1 3.8302,E2 311.3434} C_DIS
LIN {X -111.027,Y 88.1163,Z 183,A 143.7956,B 3.95,C 0.1222,E1 3.8269,E2 309.4324} C_DIS
LIN {X -113.783,Y 84.5275,Z 183,A 145.4715,B 3.9499,C 0.1273,E1 3.8241,E2 307.7777} C_DIS
LIN {X -115.6461,Y 81.9605,Z 183,A 147.0238,B 3.9499,C 0.1285,E1 3.8215,E2 306.1916} C_DIS
LIN {X -118.2518,Y 78.1537,Z 183,A 148.9223,B 3.9497,C 0.1326,E1 3.8185,E2 304.2903} C_DIS
LIN {X -120.6046,Y 74.4724,Z 183,A 150.7559,B 3.9496,C 0.1364,E1 3.8158,E2 302.4493} C_DIS
LIN {X -122.9299,Y 70.5679,Z 183,A 152.6431,B 3.9494,C 0.1405,E1 3.8131,E2 300.5572} C_DIS
LIN {X -124.7937,Y 67.216,Z 183,A 154.2884,B 3.9494,C 0.1438,E1 3.8109,E2 298.9008} C_DIS
LIN {X -126.9738,Y 62.997,Z 183,A 156.0876,B 3.9491,C 0.1493,E1 3.8087,E2 297.1187} C_DIS
LIN {X -128.4306,Y 59.9728,Z 183,A 157.576,B 3.9491,C 0.152,E1 3.8069,E2 295.6143} C_DIS
LIN {X -129.9941,Y 56.5021,Z 183,A 159.1184,B 3.9489,C 0.1559,E1 3.8051,E2 294.0727} C_DIS
LIN {X -131.2223,Y 53.5912,Z 183,A 160.5147,B 3.9488,C 0.1585,E1 3.8036,E2 292.6619} C_DIS
LIN {X -132.7159,Y 49.7733,Z 183,A 162.1214,B 3.9486,C 0.1632,E1 3.802,E2 291.0631} C_DIS
LIN {X -133.7383,Y 46.9603,Z 183,A 163.4502,B 3.9485,C 0.1657,E1 3.8008,E2 289.7198} C_DIS
LIN {X -134.9623,Y 43.3144,Z 183,A 165.0092,B 3.9483,C 0.1699,E1 3.7994,E2 288.1614} C_DIS
LIN {X -136.0314,Y 39.8293,Z 183,A 166.5559,B 3.9481,C 0.1734,E1 3.7981,E2 286.6063} C_DIS
LIN {X -137.043,Y 36.1974,Z 183,A 168.1947,B 3.948,C 0.1769,E1 3.7969,E2 284.9537} C_DIS
LIN {X -138.0853,Y 31.9936,Z 183,A 170.7895,B 3.948,C 0.1767,E1 3.7953,E2 282.2491} C_DIS
LIN {X -139.3831,Y 25.7677,Z 183,A 172.5886,B 3.9474,C 0.1884,E1 3.7943,E2 280.5539} C_DIS
LIN {X -139.868,Y 22.9788,Z 183,A 173.8927,B 3.9474,C 0.1907,E1 3.7937,E2 279.2297} C_DIS
LIN {X -140.4754,Y 18.9181,Z 183,A 175.3862,B 3.9471,C 0.1963,E1 3.7931,E2 277.7592} C_DIS
LIN {X -140.858,Y 15.8255,Z 183,A 176.8948,B 3.947,C 0.1984,E1 3.7926,E2 276.2188} C_DIS
LIN {X -141.231,Y 12.0343,Z 183,A 178.4025,B 3.9467,C 0.2029,E1 3.7923,E2 274.7165} C_DIS
LIN {X -141.4868,Y 8.5168,Z 183,A -179.9328,B 3.9466,C 0.2055,E1 3.792,E2 273.0212} C_DIS
LIN {X -141.7049,Y 3.3326,Z 183,A -177.9025,B 3.9463,C 0.2118,E1 3.7918,E2 271.0014} C_DIS
LIN {X -141.7459,Y 0.1422,Z 183,A -176.5416,B 3.9461,C 0.2151,E1 3.7918,E2 269.632} C_DIS
LIN {X -141.6957,Y -3.665,Z 183,A -174.9708,B 3.9459,C 0.2192,E1 3.7918,E2 268.0581} C_DIS
LIN {X -141.5854,Y -6.6917,Z 183,A -173.4806,B 3.9458,C 0.2211,E1 3.792,E2 266.5334} C_DIS
LIN {X -141.2367,Y -11.9663,Z 183,A -171.1004,B 3.9455,C 0.2256,E1 3.7926,E2 264.1222} C_DIS
LIN {X -140.8429,Y -15.9661,Z 183,A -169.6956,B 3.9452,C 0.2315,E1 3.793,E2 262.7478} C_DIS
LIN {X -140.3475,Y -19.8391,Z 183,A -168.1382,B 3.9449,C 0.2361,E1 3.7936,E2 261.1941} C_DIS
LIN {X -139.7159,Y -23.8903,Z 183,A -165.9196,B 3.9449,C 0.2373,E1 3.7946,E2 258.9016} C_DIS
LIN {X -138.878,Y -28.3526,Z 183,A -164.5608,B 3.9443,C 0.2452,E1 3.7953,E2 257.6076} C_DIS
LIN {X -138.1263,Y -31.8141,Z 183,A -163.0395,B 3.9441,C 0.2486,E1 3.7963,E2 256.0752} C_DIS
LIN {X -137.1584,Y -35.7649,Z 183,A -161.335,B 3.9439,C 0.2527,E1 3.7974,E2 254.3637} C_DIS
LIN {X -136.1181,Y -39.5332,Z 183,A -159.7647,B 3.9436,C 0.2571,E1 3.7986,E2 252.7955} C_DIS
LIN {X -135.2169,Y -42.5171,Z 183,A -158.4665,B 3.9434,C 0.2602,E1 3.7997,E2 251.4929} C_DIS
LIN {X -133.6921,Y -47.0938,Z 183,A -156.3964,B 3.9431,C 0.2647,E1 3.8016,E2 249.4078} C_DIS
LIN {X -132.203,Y -51.1206,Z 183,A -154.5649,B 3.9428,C 0.2686,E1 3.8034,E2 247.5642} C_DIS
LIN {X -130.8589,Y -54.4688,Z 183,A -153.0582,B 3.9426,C 0.2721,E1 3.805,E2 246.0518} C_DIS
LIN {X -129.4634,Y -57.7074,Z 183,A -151.4627,B 3.9424,C 0.2746,E1 3.8068,E2 244.434} C_DIS
LIN {X -127.3952,Y -62.1428,Z 183,A -149.5354,B 3.942,C 0.2799,E1 3.8091,E2 242.5145} C_DIS
LIN {X -125.672,Y -65.5558,Z 183,A -148.1595,B 3.9417,C 0.2848,E1 3.8108,E2 241.162} C_DIS
LIN {X -124.2112,Y -68.2877,Z 183,A -146.5681,B 3.9417,C 0.2857,E1 3.813,E2 239.5255} C_DIS
LIN {X -122.0101,Y -72.1466,Z 183,A -144.7317,B 3.9413,C 0.2897,E1 3.8156,E2 237.6843} C_DIS
LIN {X -119.7395,Y -75.8548,Z 183,A -142.9173,B 3.941,C 0.2935,E1 3.8183,E2 235.8629} C_DIS
LIN {X -117.1469,Y -79.8011,Z 183,A -140.9228,B 3.9408,C 0.2973,E1 3.8214,E2 233.8574} C_DIS
LIN {X -114.4532,Y -83.6184,Z 183,A -138.9829,B 3.9405,C 0.3012,E1 3.8246,E2 231.9111} C_DIS
LIN {X -111.665,Y -87.3067,Z 183,A -137.0826,B 3.9402,C 0.305,E1 3.8278,E2 230.007} C_DIS
LIN {X -108.8042,Y -90.8471,Z 183,A -135.1709,B 3.9399,C 0.3084,E1 3.8312,E2 228.086} C_DIS
LIN {X -105.7913,Y -94.3384,Z 183,A -133.2901,B 3.9396,C 0.3121,E1 3.8347,E2 226.2034} C_DIS
LIN {X -102.7394,Y -97.6535,Z 183,A -131.5438,B 3.9393,C 0.3163,E1 3.838,E2 224.4677} C_DIS
LIN {X -100.2741,Y -100.1833,Z 183,A -129.8873,B 3.9392,C 0.3174,E1 3.8413,E2 222.7803} C_DIS
LIN {X -96.8369,Y -103.5092,Z 183,A -127.9469,B 3.9389,C 0.3209,E1 3.8453,E2 220.8392} C_DIS
LIN {X -93.5511,Y -106.4886,Z 183,A -126.1387,B 3.9386,C 0.324,E1 3.849,E2 219.0292} C_DIS
LIN {X -90.1242,Y -109.4038,Z 183,A -124.2663,B 3.9384,C 0.3268,E1 3.8531,E2 217.1496} C_DIS
LIN {X -86.4908,Y -112.2986,Z 183,A -122.2698,B 3.9382,C 0.3289,E1 3.8575,E2 215.1369} C_DIS
Enddeposition()
END
